FUNCTION_BLOCK "Assembler_devic"   // FB1, GRAPH
{ S7_Optimized_Access := 'FALSE' }
VERSION : 0.1
   VAR_INPUT
      OFF_SQ : Bool := false;   // Turn sequence off
      INIT_SQ : Bool := false;   // Set sequence to initial state
      ACK_EF : Bool := false;   // Acknowledge all errors and faults
      S_PREV : Bool := false;   // Output previous step in parameter S_NO
      S_NEXT : Bool := false;   // Indicate next step in parameter S_NO
      SW_AUTO : Bool := false;   // Automatic mode
      SW_TAP : Bool := false;   // Semiautomatic/switch with transition
      SW_TOP : Bool := false;   // Semiautomatic/ignore transition
      SW_MAN : Bool := false;   // Manual mode
      S_SEL : Int := 0;   // Select step to be output to S_NO
      S_ON : Bool := false;   // Activate step indicated in S_NO
      S_OFF : Bool := false;   // Deactivate step indicated S_NO
      T_PUSH : Bool := false;   // Enable transition to switch in semi automatic mode
   END_VAR
   VAR_OUTPUT
      S_NO : Int := 0;   // Step number
      S_MORE : Bool := false;   // More steps are available and can be shown in S_NO
      S_ACTIVE : Bool := false;   // Step indicated in S_NO is active
      ERR_FLT : Bool := false;   // Interlock or supervision group error
      AUTO_ON : Bool := false;   // Automatic mode is active
      TAP_ON : Bool := false;   // Semiautomatic mode/step with transition enabled
      TOP_ON : Bool := false;   // Semiautomatic mode/ignore transition enabled
      MAN_ON : Bool := false;   // Manual mode is active
   END_VAR
   VAR_IN_OUT
      "assembler x set point" : Real;
      "assembler x set point value" : Real;
      "assembler z set point" : Real;
      "assembler z set point value" : Real;
      "assembler grab" : Bool;
      "assembler grabed" : Bool;
      "lid clamp" : Bool;
      "base clamp" : Bool;
      "lid clamped" : Bool;
      "base clamped" : Bool;
      "base rise" : Bool;
      "base limit" : Bool;
      "line1  ready" : Bool;
      "line2  ready" : Bool;
      "assembler rotate" : Bool;
      "assembler rotating" : Bool;
      "assembler complete" : Bool;
   END_VAR
   VAR
      SWITCH : Array[0..0] of DWord;
      SW_SQTS : Array[0..14] of Byte;
      SW_ADDR : Word := 16#1C;
      G7T_0 : GraphTransition;
      G7S_0 : GraphStep;
      PRE_CRIT : Array[0..0] of DWord;
      POST_CRIT : Array[0..0] of DWord;
      TVX : Array[0..4] of Byte;
      TTX : Array[0..4] of Byte;
      TSX : Array[0..4] of Byte;
      S00X : Array[0..4] of Byte;
      SOFFX : Array[0..4] of Byte;
      SONX : Array[0..4] of Byte;
      SAX : Array[0..4] of Byte;
      SERRX : Array[0..15] of Byte;
      SMX : Array[0..15] of Byte;
      S0X : Array[0..15] of Byte;
      S1X : Array[0..15] of Byte;
      S_DISPLAY : Int;   // Internal display of output parameter S_NO
      S_SEL_OLD : Int;   // Previous value in S_SEL
      S_DISPIDX : Byte;   // Index of the step in S_NO
      T_DISPIDX : Byte;   // Index of the transition displayed in T_NO
      MOPEDGE : Struct
         AUTO : Bool := false;
         MAN : Bool := false;
         TAP : Bool := false;
         TOP : Bool := false;
         ACK_S : Bool := false;
         REG_S : Bool := false;
         T_PREV : Bool := false;
         T_NEXT : Bool := false;
         LOCK : Bool := false;
         SUP : Bool := false;
         ACKREQ : Bool := false;
         SSKIP : Bool := false;
         OFF : Bool := false;
         INIT : Bool := false;
         HALT : Bool := false;
         TMS_HALT : Bool := false;
         OPS_ZERO : Bool := false;
         SACT_DISP : Bool := false;
         SEF_DISP : Bool := false;
         SALL_DISP : Bool := false;
         S_PREV : Bool := false;
         S_NEXT : Bool := false;
         S_SELOK : Bool := false;
         S_ON : Bool := false;
         S_OFF : Bool := false;
         T_PUSH : Bool := false;
         REG : Bool := false;
         ACK : Bool := false;
         IL_PERM : Bool := false;
         T_PERM : Bool := false;
         ILP_MAN : Bool := false;
      END_STRUCT;
      MOP : Struct   // Mode
         AUTO : Bool := true;   // Status: automatic mode
         MAN : Bool := false;   // Status: manual mode
         TAP : Bool := false;   // Status: semi automatic/switch with transition
         TOP : Bool := false;   // Status: semi automatic/ignore transition
         ACK_S : Bool := false;   // Request: acknowledge step at parameter S_NO
         REG_S : Bool := false;   // Request: register step indicated in S_NO
         T_PREV : Bool := false;   // Request: output previous valid transition in T_NO
         T_NEXT : Bool := false;   // Request: output next valid transition in T_NO
         LOCK : Bool := true;   // Status: interlocks activated
         SUP : Bool := true;   // Status: supervisions activated
         ACKREQ : Bool := true;   // Status: acknowledgment required
         SSKIP : Bool := false;   // Status: "Skip steps" enabled
         OFF : Bool := false;   // Request: deactivate all steps
         INIT : Bool := true;   // Request: set sequence to initial state
         HALT : Bool := false;   // Status: sequence halted
         TMS_HALT : Bool := false;   // Status: all internal timers held
         OPS_ZERO : Bool := false;   // Status: set all operands processed with N, L, D instructions to 0
         SACT_DISP : Bool := true;   // Status: display active steps only
         SEF_DISP : Bool := false;   // Status: display only steps with errors and disrupted steps
         SALL_DISP : Bool := false;   // Status: display all steps
         S_PREV : Bool := false;   // Request: output previous step to S_NO
         S_NEXT : Bool := false;   // Request: Output next step at S_NO parameter
         S_SELOK : Bool := false;   // Request: output step number from S_SEL to S_NO
         S_ON : Bool := false;   // Request: activate step indicated in S_NO
         S_OFF : Bool := false;   // Request: deactivate step at parameter S_NO
         T_PUSH : Bool := false;   // Request: transition switching enabled
         REG : Bool := false;   // Request: register all interlock and supervision errors
         ACK : Bool := false;   // Request: acknowledge all interlock and supervision errors
         IL_PERM : Bool := false;   // Status: permanent processing of all interlocks
         T_PERM : Bool := false;   // Status: permanent processing of all transitions
         ILP_MAN : Bool := false;   // Status: permanent processing of all interlocks in manual mode
      END_STRUCT;
      TICKS : Struct   // Clock speeds
         DELTA : Time := T#0ms;   // Time difference between cycles
         OLD : Time := T#0ms;   // 10 ms clock counter value in last cycle
         NEW : Time := T#0ms;   // 10 ms clock counter value in this cycle
      END_STRUCT;
      SQ_FLAGS : Struct   // Sequence bit memory
         ERR_FLT : Bool := false;   // Interlock and supervision group error
         ERROR : Bool := false;   // Interlock group error
         FAULT : Bool := false;   // Supervision group error
         RT_FAIL : Bool := false;   // Runtime error
         NO_SNO : Bool := false;   // Requested step number not found
         NF_OFL : Bool := false;   // Overflow: too many ON or OFF requests
         SA_OFL : Bool := false;   // Overflow: too many steps active
         TV_OFL : Bool := false;   // Overflow: too many valid transitions
         MSG_OFL : Bool := false;   // Overflow: not enough system resources for ALARM_S
         NO_SWI : Bool := false;   // Do not switch in this cycle
         CYC_OP : Bool := false;   // Cyclic execution of the sequence after initialization
         AS_MSG : Bool := true;   // Alarms during runtime enabled or disabled by instruction
         AS_SEND : Bool := false;   // Send alarms from WR_USMSG or only enter in diagnostics buffer
         SQ_BUSY : Bool := false;   // Internal edge bit memory for sequence processing
         SA_BUSY : Bool := false;   // Internal edge bit memory for sequence processing
         AS_SIG : Bool := false;   // Edge bit memory for alarms from Alarm_S and Alarm_SQ
      END_STRUCT;
      S_PTR : DWord := 16#890;
      S_PTR2 : DWord := 16#0;
      S_PTR3 : DWord := 16#1AA0;
      S_PTR4 : DWord := 16#1A20;
      T_PTR : DWord := 16#19A0;
      C_AR2 : DWord := 16#0;
      M_FBDB : DWord := 16#10000;
      M_SNO : Word := 16#0;
      M_EVID : Word := 16#0;
      M_EVIL : C_Alarm_s;
      M_EVSV : C_Alarm_s;
      M_EV : DWord := 16#1890;
      CRIT : Array[0..31] of Bool;
      S_START : Byte := 16#0;
      S_IDX : Byte := 16#0;
      S_INT : Int := 72;
      S_TMP : Byte := 16#0;
      T_START : Byte := 16#0;
      T_IDX : Byte := 16#0;
      T_TMP : Byte := 16#0;
      T_TMP2 : Byte := 16#00;
      TV_POT : Byte := 16#06;
      RETURN1 : Byte := 16#0;
      RETURN2 : Byte := 16#0;
      SINI : Array[0..4] of Byte;
      LSTT : Array[0..13] of Byte;
      ATAJ : Array[0..13] of Byte;
      ATAB : Array[0..13] of Byte;
      PSTT : Array[0..13] of Byte;
      NSTT : Array[0..13] of Byte;
      ASSJ : Array[0..14] of Byte;
      ASSB : Array[0..14] of Byte;
      PTTS : Array[0..14] of Byte;
      NTTS : Array[0..14] of Byte;
      PRE_CNT : Word := 16#1;
      POST_CNT : Word := 16#1;
      ADR_COND : Word := 16#0;
      MAX_TVAL : Byte := 16#3;
      MAX_SACT : Byte := 16#3;
      MAX_CRIT : Byte := 16#4;
      T_CNT : Byte := 16#D;
      SUP_CNT : Byte := 16#0;
      LOCK_CNT : Byte;
      S_CNT : Byte := 16#E;
      SQ_CNT : Byte := 16#1;
      PRS_INPAR : DWord := 16#E000FEC8;
      PRS_OUTPAR : DWord := 16#E000800F;
      GC_FLAGS : Struct
         T_MACH : Byte := 16#EB;
         COND_ED : Byte := 16#E3;
         W_LEVEL : Byte := 16#D5;
         FB_IF : Byte := 16#FA;
         AS_MSG : Word := 16#404;
         SSB : Word := 16#108;
         DILG : Word := 16#470;
         ADDR_T0 : Word := 16#32;
         CRIT_AVAIL : Bool := false;
         SSKIP_AVAIL : Bool := true;
         SSKIP_ON : Bool := false;
         ACK_REQ : Bool := true;
         SYNC_AVAIL : Bool := true;
         ILP_MAN : Bool := false;
         SWM_LOCKED : Bool := false;
         SAVE_SW : Bool := true;
      END_STRUCT;
      G7_FBMARK : Byte := 16#3C;
      G7_RELEASE : Byte := 16#3C;
      G7_ID2 : Byte := 16#37;
      G7_ID1 : Byte := 16#47;
   END_VAR
   // SW_SQTS[0] := 16#4;
   // SWITCH[0] := 16#40020000;
   // SW_SQTS[2] := 16#1;
   // SW_SQTS[3] := 16#1;
   // SW_SQTS[4] := 16#2;
   // SW_SQTS[5] := 16#2;
   // SW_SQTS[6] := 16#2;
   // SW_SQTS[7] := 16#3;
   // TVX[0] := 16#1;
   // TTX[0] := 16#1;
   // TSX[0] := 16#1;
   // S00X[0] := 16#1;
   // SOFFX[0] := 16#1;
   // SONX[0] := 16#1;
   // SAX[0] := 16#1;
   // SERRX[0] := 16#1;
   // SMX[0] := 16#1;
   // S0X[0] := 16#1;
   // S1X[0] := 16#1;
   // SINI[0] := 16#2;
   // SINI[1] := 16#1;
   // SINI[2] := 0;
   // SINI[3] := 0;
   // SINI[4] := 0;
   // LSTT[0] := 0;
   // LSTT[1] := 0;
   // LSTT[2] := 0;
   // LSTT[3] := 0;
   // LSTT[4] := 0;
   // LSTT[5] := 0;
   // LSTT[6] := 0;
   // LSTT[7] := 0;
   // ATAJ[0] := 0;
   // ATAJ[1] := 16#1;
   // ATAJ[2] := 16#2;
   // ATAJ[3] := 16#3;
   // ATAJ[4] := 16#4;
   // ATAJ[5] := 16#5;
   // ATAJ[6] := 16#6;
   // ATAJ[7] := 16#7;
   // ATAB[0] := 0;
   // ATAB[1] := 16#1;
   // ATAB[2] := 16#2;
   // ATAB[3] := 16#3;
   // ATAB[4] := 16#4;
   // ATAB[5] := 16#5;
   // ATAB[6] := 16#6;
   // ATAB[7] := 16#7;
   // PSTT[0] := 0;
   // PSTT[1] := 16#1;
   // PSTT[2] := 16#2;
   // PSTT[3] := 16#3;
   // PSTT[4] := 16#4;
   // PSTT[5] := 16#5;
   // PSTT[6] := 16#8;
   // PSTT[7] := 16#9;
   // NSTT[0] := 16#1;
   // NSTT[1] := 16#2;
   // NSTT[2] := 16#3;
   // NSTT[3] := 16#8;
   // NSTT[5] := 16#6;
   // NSTT[6] := 16#9;
   // NSTT[7] := 16#A;
   // ASSJ[0] := 0;
   // ASSJ[1] := 16#1;
   // ASSJ[2] := 16#2;
   // ASSJ[3] := 16#6;
   // ASSJ[4] := 16#4;
   // ASSJ[5] := 16#5;
   // ASSJ[6] := 16#3;
   // ASSJ[7] := 16#7;
   // ASSB[0] := 0;
   // ASSB[1] := 16#1;
   // ASSB[2] := 16#4;
   // ASSB[3] := 16#3;
   // ASSB[4] := 16#2;
   // ASSB[5] := 16#5;
   // ASSB[6] := 16#6;
   // ASSB[7] := 16#7;
   // PTTS[0] := 0;
   // PTTS[2] := 16#1;
   // PTTS[3] := 16#2;
   // PTTS[4] := 16#1;
   // PTTS[5] := 16#4;
   // PTTS[6] := 16#5;
   // PTTS[7] := 16#8;
   // NTTS[0] := 0;
   // NTTS[1] := 16#1;
   // NTTS[2] := 16#2;
   // NTTS[3] := 16#3;
   // NTTS[4] := 16#4;
   // NTTS[5] := 16#5;
   // NTTS[6] := 16#3;
   // NTTS[7] := 16#9;
   // SW_SQTS[8] := 16#3;
   // NTTS[14] := 16#D;
   // PTTS[14] := 16#C;
   // PTTS[13] := 16#B;
   // ASSB[14] := 16#E;
   // ASSB[13] := 16#D;
   // ASSJ[14] := 16#E;
   // ASSJ[13] := 16#D;
   // NSTT[13] := 16#1;
   // NSTT[12] := 16#E;
   // PSTT[13] := 16#E;
   // ATAB[13] := 16#D;
   // ATAB[12] := 16#C;
   // ATAJ[13] := 16#D;
   // ATAJ[12] := 16#C;
   // LSTT[13] := 16#1;
   // LSTT[12] := 0;
   // SW_SQTS[14] := 16#3;
   // SW_SQTS[13] := 16#3;
   // NSTT[4] := 16#5;
   // NTTS[12] := 16#B;
   // NTTS[11] := 16#A;
   // NTTS[10] := 16#8;
   // NTTS[9] := 16#7;
   // PTTS[12] := 16#A;
   // PTTS[11] := 16#9;
   // PTTS[10] := 16#7;
   // ASSJ[8] := 16#8;
   // ASSB[12] := 16#C;
   // ASSB[11] := 16#B;
   // ASSB[10] := 16#A;
   // ASSB[9] := 16#9;
   // ASSJ[12] := 16#C;
   // ASSJ[11] := 16#B;
   // ASSJ[10] := 16#A;
   // ASSJ[9] := 16#9;
   // NSTT[11] := 16#D;
   // ASSB[8] := 16#8;
   // NSTT[9] := 16#B;
   // NSTT[8] := 16#7;
   // PSTT[11] := 16#C;
   // PSTT[10] := 16#B;
   // PSTT[9] := 16#7;
   // PSTT[8] := 16#A;
   // ATAB[11] := 16#B;
   // ATAB[10] := 16#A;
   // ATAB[9] := 16#9;
   // PTTS[8] := 16#3;
   // ATAJ[11] := 16#B;
   // ATAJ[10] := 16#A;
   // ATAJ[9] := 16#9;
   // ATAJ[8] := 16#8;
   // LSTT[11] := 0;
   // LSTT[10] := 0;
   // LSTT[9] := 0;
   // LSTT[8] := 0;
   // SW_SQTS[12] := 16#3;
   // NTTS[8] := 16#6;
   // SW_SQTS[10] := 16#3;
   // SW_SQTS[9] := 16#3;
   // ATAB[8] := 16#8;
   // NSTT[10] := 16#C;
   // PTTS[9] := 16#6;
   // PSTT[12] := 16#D;
   // NTTS[13] := 16#C;
   // SW_SQTS[11] := 16#3;
BEGIN
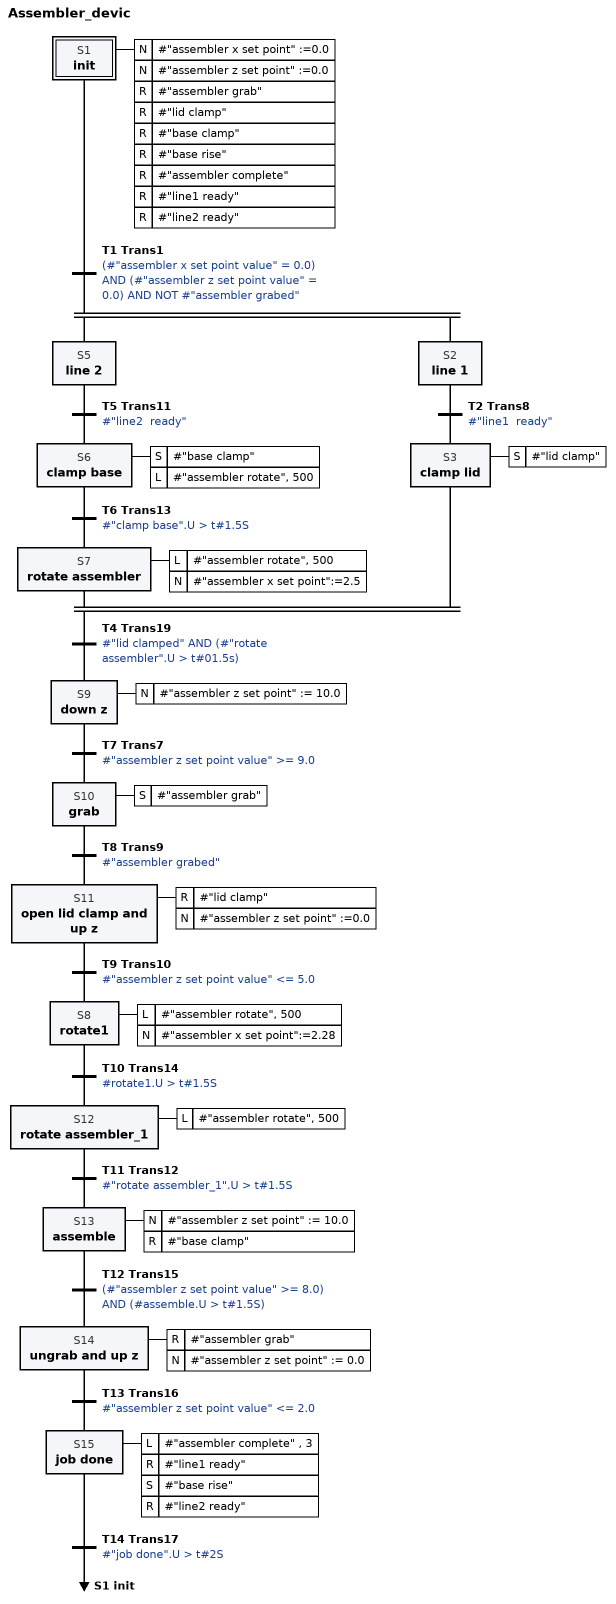
   // sequencer 1
   INITIAL_STEP init:   // S1
              N    #"assembler x set point" :=0.0
              N    #"assembler z set point" :=0.0
              R    #"assembler grab"
              R    #"lid clamp"
              R    #"base clamp"
              R    #"base rise"
              R    #"assembler complete"
              R    #"line1  ready"
              R    #"line2  ready"
   END_STEP
   TRANSITION Trans1 FROM init TO ("line 2", "line 1")   // T1
      := (#"assembler x set point value" = 0.0) AND (#"assembler z set point value" = 0.0) AND NOT #"assembler grabed";
   END_TRANSITION
   STEP "clamp lid":   // S3
              S    #"lid clamp"
   END_STEP
   STEP "line 2":   // S5
   END_STEP
   TRANSITION Trans11 FROM "line 2" TO "clamp base"   // T5
      := #"line2  ready";
   END_TRANSITION
   STEP "line 1":   // S2
   END_STEP
   TRANSITION Trans8 FROM "line 1" TO "clamp lid"   // T2
      := #"line1  ready";
   END_TRANSITION
   STEP grab:   // S10
              S    #"assembler grab"
   END_STEP
   TRANSITION Trans9 FROM grab TO "open lid clamp and up z"   // T8
      := #"assembler grabed";
   END_TRANSITION
   STEP "clamp base":   // S6
              S    #"base clamp"
              L    #"assembler rotate", 500
   END_STEP
   TRANSITION Trans13 FROM "clamp base" TO "rotate assembler"   // T6
      := #"clamp base".U > t#1.5S;
   END_TRANSITION
   STEP "rotate assembler":   // S7
              L    #"assembler rotate", 500
              N    #"assembler x set point":=2.5
   END_STEP
   TRANSITION Trans19 FROM ("clamp lid", "rotate assembler") TO "down z"   // T4
      := #"lid clamped" AND (#"rotate assembler".U > t#01.5s);
   END_TRANSITION
   STEP "down z":   // S9
              N    #"assembler z set point" := 10.0
   END_STEP
   TRANSITION Trans7 FROM "down z" TO grab   // T7
      := #"assembler z set point value" >= 9.0;
   END_TRANSITION
   STEP "open lid clamp and up z":   // S11
              R    #"lid clamp"
              N    #"assembler z set point" :=0.0
   END_STEP
   TRANSITION Trans10 FROM "open lid clamp and up z" TO rotate1   // T9
      := #"assembler z set point value" <= 5.0;
   END_TRANSITION
   STEP rotate1:   // S8
              L    #"assembler rotate", 500
              N    #"assembler x set point":=2.28
   END_STEP
   TRANSITION Trans14 FROM rotate1 TO "rotate assembler_1"   // T10
      := #rotate1.U > t#1.5S;
   END_TRANSITION
   STEP "rotate assembler_1":   // S12
              L    #"assembler rotate", 500
   END_STEP
   TRANSITION Trans12 FROM "rotate assembler_1" TO assemble   // T11
      := #"rotate assembler_1".U > t#1.5S;
   END_TRANSITION
   STEP assemble:   // S13
              N    #"assembler z set point" := 10.0
              R    #"base clamp"
   END_STEP
   TRANSITION Trans15 FROM assemble TO "ungrab and up z"   // T12
      := (#"assembler z set point value" >= 8.0) AND (#assemble.U > t#1.5S);
   END_TRANSITION
   STEP "ungrab and up z":   // S14
              R    #"assembler grab"
              N    #"assembler z set point" := 0.0
   END_STEP
   TRANSITION Trans16 FROM "ungrab and up z" TO "job done"   // T13
      := #"assembler z set point value" <= 2.0;
   END_TRANSITION
   STEP "job done":   // S15
              L    #"assembler complete" , 3
              R    #"line1  ready"
              S    #"base rise"
              R    #"line2  ready"
   END_STEP
   TRANSITION Trans17 FROM "job done" TO init   // T14, jump
      := #"job done".U > t#2S;
   END_TRANSITION
END_FUNCTION_BLOCK

FUNCTION "Assembler" : Void   // FC4, LAD
{ S7_Optimized_Access := 'FALSE' }
VERSION : 0.1
BEGIN

REGION Network 1: Control Convoyers
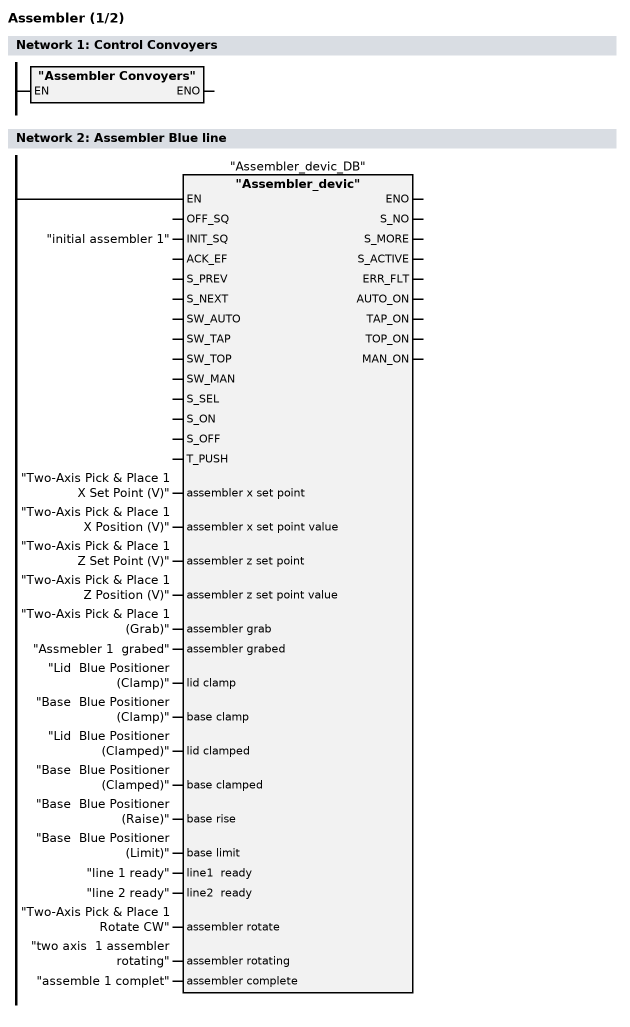
   RUNG wire#powerrail
      "Assembler Convoyers"()
   END_RUNG
   // the same network as SCL:
   "Assembler Convoyers"();
END_REGION

REGION Network 2: Assembler Blue line
   RUNG wire#powerrail
      "Assembler_devic_DB"(OFF_SQ :=, INIT_SQ := "initial assembler 1", ACK_EF :=, S_PREV :=, S_NEXT :=, SW_AUTO :=, SW_TAP :=, SW_TOP :=, SW_MAN :=, S_SEL :=, S_ON :=, S_OFF :=, T_PUSH :=, "assembler x set point" := "Two-Axis Pick & Place 1 X Set Point (V)", "assembler x set point value" := "Two-Axis Pick & Place 1 X Position (V)", "assembler z set point" := "Two-Axis Pick & Place 1 Z Set Point (V)", "assembler z set point value" := "Two-Axis Pick & Place 1 Z Position (V)", "assembler grab" := "Two-Axis Pick & Place 1 (Grab)", "assembler grabed" := "Assmebler 1  grabed", "lid clamp" := "Lid  Blue Positioner (Clamp)", "base clamp" := "Base  Blue Positioner (Clamp)", "lid clamped" := "Lid  Blue Positioner (Clamped)", "base clamped" := "Base  Blue Positioner (Clamped)", "base rise" := "Base  Blue Positioner  (Raise)", "base limit" := "Base  Blue Positioner (Limit)", "line1  ready" := "line 1 ready", "line2  ready" := "line 2 ready", "assembler rotate" := "Two-Axis Pick & Place 1 Rotate CW", "assembler rotating" := "two axis  1 assembler rotating", "assembler complete" := "assemble 1 complet", S_NO =>, S_MORE =>, S_ACTIVE =>, ERR_FLT =>, AUTO_ON =>, TAP_ON =>, TOP_ON =>, MAN_ON =>)
   END_RUNG
   // the same network as SCL:
   "Assembler_devic_DB"(INIT_SQ := "initial assembler 1",   // "Assembler_devic"
                        "assembler x set point" := "Two-Axis Pick & Place 1 X Set Point (V)",
                        "assembler x set point value" := "Two-Axis Pick & Place 1 X Position (V)",
                        "assembler z set point" := "Two-Axis Pick & Place 1 Z Set Point (V)",
                        "assembler z set point value" := "Two-Axis Pick & Place 1 Z Position (V)",
                        "assembler grab" := "Two-Axis Pick & Place 1 (Grab)",
                        "assembler grabed" := "Assmebler 1  grabed",
                        "lid clamp" := "Lid  Blue Positioner (Clamp)",
                        "base clamp" := "Base  Blue Positioner (Clamp)",
                        "lid clamped" := "Lid  Blue Positioner (Clamped)",
                        "base clamped" := "Base  Blue Positioner (Clamped)",
                        "base rise" := "Base  Blue Positioner  (Raise)",
                        "base limit" := "Base  Blue Positioner (Limit)",
                        "line1  ready" := "line 1 ready",
                        "line2  ready" := "line 2 ready",
                        "assembler rotate" := "Two-Axis Pick & Place 1 Rotate CW",
                        "assembler rotating" := "two axis  1 assembler rotating",
                        "assembler complete" := "assemble 1 complet");
END_REGION

REGION Network 3: Assembler green line
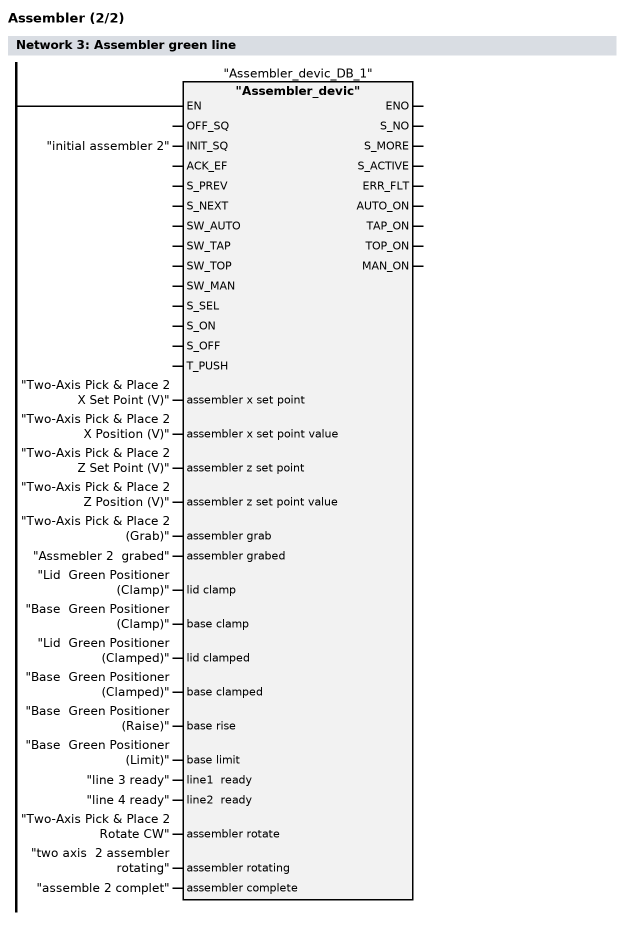
   RUNG wire#powerrail
      "Assembler_devic_DB_1"(OFF_SQ :=, INIT_SQ := "initial assembler 2", ACK_EF :=, S_PREV :=, S_NEXT :=, SW_AUTO :=, SW_TAP :=, SW_TOP :=, SW_MAN :=, S_SEL :=, S_ON :=, S_OFF :=, T_PUSH :=, "assembler x set point" := "Two-Axis Pick & Place 2 X Set Point (V)", "assembler x set point value" := "Two-Axis Pick & Place 2 X Position (V)", "assembler z set point" := "Two-Axis Pick & Place 2 Z Set Point (V)", "assembler z set point value" := "Two-Axis Pick & Place 2 Z Position (V)", "assembler grab" := "Two-Axis Pick & Place 2 (Grab)", "assembler grabed" := "Assmebler 2  grabed", "lid clamp" := "Lid  Green Positioner (Clamp)", "base clamp" := "Base  Green Positioner (Clamp)", "lid clamped" := "Lid  Green Positioner (Clamped)", "base clamped" := "Base  Green Positioner (Clamped)", "base rise" := "Base  Green Positioner (Raise)", "base limit" := "Base  Green Positioner (Limit)", "line1  ready" := "line 3 ready", "line2  ready" := "line 4 ready", "assembler rotate" := "Two-Axis Pick & Place 2 Rotate CW", "assembler rotating" := "two axis  2 assembler rotating", "assembler complete" := "assemble 2 complet", S_NO =>, S_MORE =>, S_ACTIVE =>, ERR_FLT =>, AUTO_ON =>, TAP_ON =>, TOP_ON =>, MAN_ON =>)
   END_RUNG
   // the same network as SCL:
   "Assembler_devic_DB_1"(INIT_SQ := "initial assembler 2",   // "Assembler_devic"
                          "assembler x set point" := "Two-Axis Pick & Place 2 X Set Point (V)",
                          "assembler x set point value" := "Two-Axis Pick & Place 2 X Position (V)",
                          "assembler z set point" := "Two-Axis Pick & Place 2 Z Set Point (V)",
                          "assembler z set point value" := "Two-Axis Pick & Place 2 Z Position (V)",
                          "assembler grab" := "Two-Axis Pick & Place 2 (Grab)",
                          "assembler grabed" := "Assmebler 2  grabed",
                          "lid clamp" := "Lid  Green Positioner (Clamp)",
                          "base clamp" := "Base  Green Positioner (Clamp)",
                          "lid clamped" := "Lid  Green Positioner (Clamped)",
                          "base clamped" := "Base  Green Positioner (Clamped)",
                          "base rise" := "Base  Green Positioner (Raise)",
                          "base limit" := "Base  Green Positioner (Limit)",
                          "line1  ready" := "line 3 ready",
                          "line2  ready" := "line 4 ready",
                          "assembler rotate" := "Two-Axis Pick & Place 2 Rotate CW",
                          "assembler rotating" := "two axis  2 assembler rotating",
                          "assembler complete" := "assemble 2 complet");
END_REGION
END_FUNCTION

FUNCTION "Sort" : Void   // FC5, LAD
{ S7_Optimized_Access := 'FALSE' }
VERSION : 0.1
BEGIN

REGION Network 1: Blue Lid
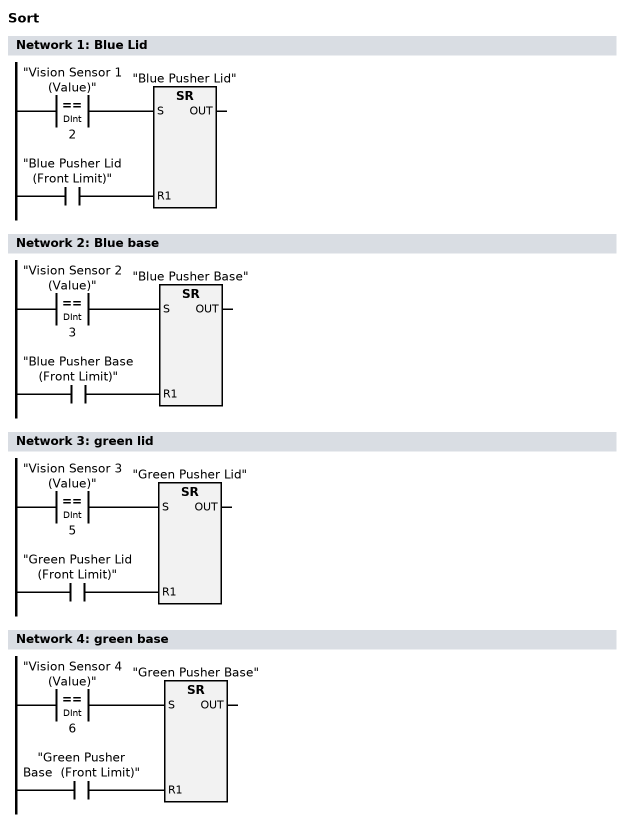
   RUNG wire#powerrail
      { S7_Templates := "SrcType := DInt" } EQ_Contact(in1 := "Vision Sensor 1 (Value)", in2 := 2)
      S_SR(operand := "Blue Pusher Lid", r1 := wire#w1)
   END_RUNG
   RUNG wire#powerrail
      Contact( "Blue Pusher Lid (Front Limit)" )
   END_RUNG wire#w1
   // the same network as SCL:
   IF "Vision Sensor 1 (Value)" = 2 THEN
       "Blue Pusher Lid" := TRUE;   // SR flip-flop
   END_IF;
   IF "Blue Pusher Lid (Front Limit)" THEN "Blue Pusher Lid" := FALSE; END_IF;
END_REGION

REGION Network 2: Blue base
   RUNG wire#powerrail
      { S7_Templates := "SrcType := DInt" } EQ_Contact(in1 := "Vision Sensor 2 (Value)", in2 := 3)
      S_SR(operand := "Blue Pusher Base", r1 := wire#w1)
   END_RUNG
   RUNG wire#powerrail
      Contact( "Blue Pusher Base  (Front Limit)" )
   END_RUNG wire#w1
   // the same network as SCL:
   IF "Vision Sensor 2 (Value)" = 3 THEN
       "Blue Pusher Base" := TRUE;   // SR flip-flop
   END_IF;
   IF "Blue Pusher Base  (Front Limit)" THEN "Blue Pusher Base" := FALSE; END_IF;
END_REGION

REGION Network 3: green lid
   RUNG wire#powerrail
      { S7_Templates := "SrcType := DInt" } EQ_Contact(in1 := "Vision Sensor 3 (Value)", in2 := 5)
      S_SR(operand := "Green Pusher Lid", r1 := wire#w1)
   END_RUNG
   RUNG wire#powerrail
      Contact( "Green Pusher Lid (Front Limit)" )
   END_RUNG wire#w1
   // the same network as SCL:
   IF "Vision Sensor 3 (Value)" = 5 THEN
       "Green Pusher Lid" := TRUE;   // SR flip-flop
   END_IF;
   IF "Green Pusher Lid (Front Limit)" THEN "Green Pusher Lid" := FALSE; END_IF;
END_REGION

REGION Network 4: green base
   RUNG wire#powerrail
      { S7_Templates := "SrcType := DInt" } EQ_Contact(in1 := "Vision Sensor 4 (Value)", in2 := 6)
      S_SR(operand := "Green Pusher Base", r1 := wire#w1)
   END_RUNG
   RUNG wire#powerrail
      Contact( "Green Pusher Base  (Front Limit)" )
   END_RUNG wire#w1
   // the same network as SCL:
   IF "Vision Sensor 4 (Value)" = 6 THEN
       "Green Pusher Base" := TRUE;   // SR flip-flop
   END_IF;
   IF "Green Pusher Base  (Front Limit)" THEN "Green Pusher Base" := FALSE; END_IF;
END_REGION
END_FUNCTION

FUNCTION "Assembler Convoyers" : Void   // FC6, LAD
{ S7_Optimized_Access := 'FALSE' }
VERSION : 0.1
   VAR_TEMP   // added for the SCL form of the ladder/FBD networks
      _w1 : Bool;
      _w2 : Bool;
      _w3 : Bool;
   END_VAR
BEGIN

REGION Network 1: Blue lid Convoyer *
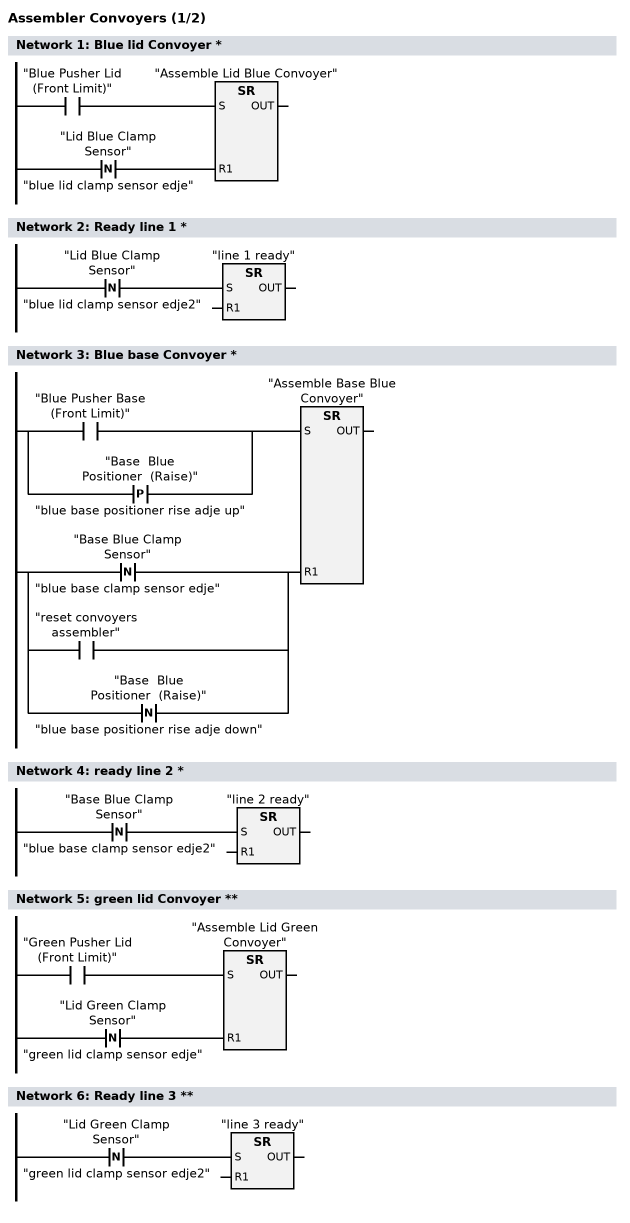
   RUNG wire#powerrail
      Contact( "Blue Pusher Lid (Front Limit)" )
      S_SR(operand := "Assemble Lid Blue Convoyer", r1 := wire#w1)
   END_RUNG
   RUNG wire#powerrail
      N_Contact(operand := "Lid Blue Clamp Sensor", bit := "blue lid clamp sensor edje")
   END_RUNG wire#w1
   // the same network as SCL:
   #_w1 := NOT "Lid Blue Clamp Sensor" AND "blue lid clamp sensor edje";   // falling edge of "Lid Blue Clamp Sensor"
   "blue lid clamp sensor edje" := "Lid Blue Clamp Sensor";
   IF "Blue Pusher Lid (Front Limit)" THEN
       "Assemble Lid Blue Convoyer" := TRUE;   // SR flip-flop
   END_IF;
   IF #_w1 THEN "Assemble Lid Blue Convoyer" := FALSE; END_IF;
END_REGION

REGION Network 2: Ready line 1 *
   RUNG wire#powerrail
      N_Contact(operand := "Lid Blue Clamp Sensor", bit := "blue lid clamp sensor edje2")
      S_SR(operand := "line 1 ready", r1 :=)
   END_RUNG
   // the same network as SCL:
   #_w1 := NOT "Lid Blue Clamp Sensor" AND "blue lid clamp sensor edje2";   // falling edge of "Lid Blue Clamp Sensor"
   "blue lid clamp sensor edje2" := "Lid Blue Clamp Sensor";
   IF #_w1 THEN
       "line 1 ready" := TRUE;   // SR flip-flop
   END_IF;
END_REGION

REGION Network 3: Blue base Convoyer *
   RUNG wire#powerrail
      Contact( "Blue Pusher Base  (Front Limit)" )
      wire#w1
      S_SR(operand := "Assemble Base Blue Convoyer", r1 := wire#w2)
   END_RUNG
   RUNG wire#powerrail
      P_Contact(operand := "Base  Blue Positioner  (Raise)", bit := "blue base positioner rise adje up")
   END_RUNG wire#w1
   RUNG wire#powerrail
      N_Contact(operand := "Base Blue Clamp Sensor", bit := "blue base clamp sensor edje")
   END_RUNG wire#w2
   RUNG wire#powerrail
      Contact( "reset convoyers assembler" )
   END_RUNG wire#w2
   RUNG wire#powerrail
      N_Contact(operand := "Base  Blue Positioner  (Raise)", bit := "blue base positioner rise adje down")
   END_RUNG wire#w2
   // the same network as SCL:
   #_w1 := "Base  Blue Positioner  (Raise)" AND NOT "blue base positioner rise adje up";   // rising edge of "Base  Blue Positioner  (Raise)"
   "blue base positioner rise adje up" := "Base  Blue Positioner  (Raise)";
   #_w2 := NOT "Base Blue Clamp Sensor" AND "blue base clamp sensor edje";   // falling edge of "Base Blue Clamp Sensor"
   "blue base clamp sensor edje" := "Base Blue Clamp Sensor";
   #_w3 := NOT "Base  Blue Positioner  (Raise)" AND "blue base positioner rise adje down";   // falling edge of "Base  Blue Positioner  (Raise)"
   "blue base positioner rise adje down" := "Base  Blue Positioner  (Raise)";
   IF "Blue Pusher Base  (Front Limit)" OR #_w1 THEN
       "Assemble Base Blue Convoyer" := TRUE;   // SR flip-flop
   END_IF;
   IF #_w2 OR "reset convoyers assembler" OR #_w3 THEN "Assemble Base Blue Convoyer" := FALSE; END_IF;
END_REGION

REGION Network 4: ready line 2 *
   RUNG wire#powerrail
      N_Contact(operand := "Base Blue Clamp Sensor", bit := "blue base clamp sensor edje2")
      S_SR(operand := "line 2 ready", r1 :=)
   END_RUNG
   // the same network as SCL:
   #_w1 := NOT "Base Blue Clamp Sensor" AND "blue base clamp sensor edje2";   // falling edge of "Base Blue Clamp Sensor"
   "blue base clamp sensor edje2" := "Base Blue Clamp Sensor";
   IF #_w1 THEN
       "line 2 ready" := TRUE;   // SR flip-flop
   END_IF;
END_REGION

REGION Network 5: green lid Convoyer **
   RUNG wire#powerrail
      Contact( "Green Pusher Lid (Front Limit)" )
      S_SR(operand := "Assemble Lid Green Convoyer", r1 := wire#w1)
   END_RUNG
   RUNG wire#powerrail
      N_Contact(operand := "Lid Green Clamp Sensor", bit := "green lid clamp sensor edje")
   END_RUNG wire#w1
   // the same network as SCL:
   #_w1 := NOT "Lid Green Clamp Sensor" AND "green lid clamp sensor edje";   // falling edge of "Lid Green Clamp Sensor"
   "green lid clamp sensor edje" := "Lid Green Clamp Sensor";
   IF "Green Pusher Lid (Front Limit)" THEN
       "Assemble Lid Green Convoyer" := TRUE;   // SR flip-flop
   END_IF;
   IF #_w1 THEN "Assemble Lid Green Convoyer" := FALSE; END_IF;
END_REGION

REGION Network 6: Ready line 3 **
   RUNG wire#powerrail
      N_Contact(operand := "Lid Green Clamp Sensor", bit := "green lid clamp sensor edje2")
      S_SR(operand := "line 3 ready", r1 :=)
   END_RUNG
   // the same network as SCL:
   #_w1 := NOT "Lid Green Clamp Sensor" AND "green lid clamp sensor edje2";   // falling edge of "Lid Green Clamp Sensor"
   "green lid clamp sensor edje2" := "Lid Green Clamp Sensor";
   IF #_w1 THEN
       "line 3 ready" := TRUE;   // SR flip-flop
   END_IF;
END_REGION

REGION Network 7: green base Convoyer **
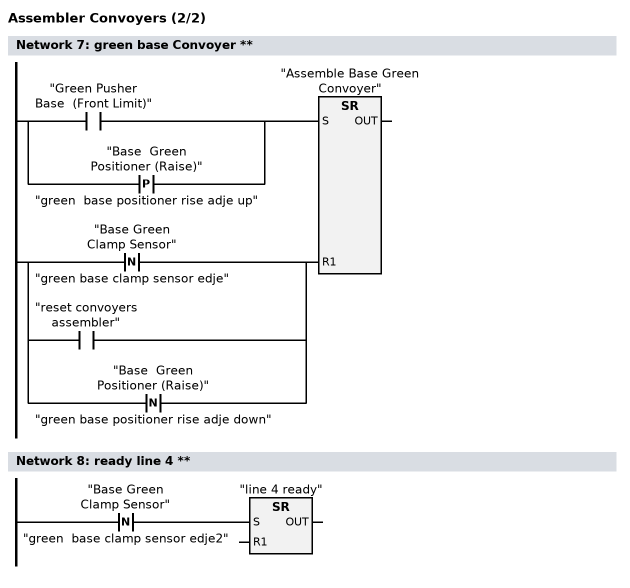
   RUNG wire#powerrail
      Contact( "Green Pusher Base  (Front Limit)" )
      wire#w1
      S_SR(operand := "Assemble Base Green Convoyer", r1 := wire#w2)
   END_RUNG
   RUNG wire#powerrail
      P_Contact(operand := "Base  Green Positioner (Raise)", bit := "green  base positioner rise adje up")
   END_RUNG wire#w1
   RUNG wire#powerrail
      N_Contact(operand := "Base Green Clamp Sensor", bit := "green base clamp sensor edje")
   END_RUNG wire#w2
   RUNG wire#powerrail
      Contact( "reset convoyers assembler" )
   END_RUNG wire#w2
   RUNG wire#powerrail
      N_Contact(operand := "Base  Green Positioner (Raise)", bit := "green base positioner rise adje down")
   END_RUNG wire#w2
   // the same network as SCL:
   #_w1 := "Base  Green Positioner (Raise)" AND NOT "green  base positioner rise adje up";   // rising edge of "Base  Green Positioner (Raise)"
   "green  base positioner rise adje up" := "Base  Green Positioner (Raise)";
   #_w2 := NOT "Base Green Clamp Sensor" AND "green base clamp sensor edje";   // falling edge of "Base Green Clamp Sensor"
   "green base clamp sensor edje" := "Base Green Clamp Sensor";
   #_w3 := NOT "Base  Green Positioner (Raise)" AND "green base positioner rise adje down";   // falling edge of "Base  Green Positioner (Raise)"
   "green base positioner rise adje down" := "Base  Green Positioner (Raise)";
   IF "Green Pusher Base  (Front Limit)" OR #_w1 THEN
       "Assemble Base Green Convoyer" := TRUE;   // SR flip-flop
   END_IF;
   IF #_w2 OR "reset convoyers assembler" OR #_w3 THEN "Assemble Base Green Convoyer" := FALSE; END_IF;
END_REGION

REGION Network 8: ready line 4 **
   RUNG wire#powerrail
      N_Contact(operand := "Base Green Clamp Sensor", bit := "green  base clamp sensor edje2")
      S_SR(operand := "line 4 ready", r1 :=)
   END_RUNG
   // the same network as SCL:
   #_w1 := NOT "Base Green Clamp Sensor" AND "green  base clamp sensor edje2";   // falling edge of "Base Green Clamp Sensor"
   "green  base clamp sensor edje2" := "Base Green Clamp Sensor";
   IF #_w1 THEN
       "line 4 ready" := TRUE;   // SR flip-flop
   END_IF;
END_REGION
END_FUNCTION

// folder: Storage System

FUNCTION_BLOCK "Turntable"   // FB4, GRAPH
{ S7_Optimized_Access := 'FALSE' }
VERSION : 0.1
   VAR_INPUT
      OFF_SQ : Bool := false;   // Turn sequence off
      INIT_SQ : Bool := false;   // Set sequence to initial state
      ACK_EF : Bool := false;   // Acknowledge all errors and faults
      S_PREV : Bool := false;   // Output previous step in parameter S_NO
      S_NEXT : Bool := false;   // Indicate next step in parameter S_NO
      SW_AUTO : Bool := false;   // Automatic mode
      SW_TAP : Bool := false;   // Semiautomatic/switch with transition
      SW_TOP : Bool := false;   // Semiautomatic/ignore transition
      SW_MAN : Bool := false;   // Manual mode
      S_SEL : Int := 0;   // Select step to be output to S_NO
      S_ON : Bool := false;   // Activate step indicated in S_NO
      S_OFF : Bool := false;   // Deactivate step indicated S_NO
      T_PUSH : Bool := false;   // Enable transition to switch in semi automatic mode
   END_VAR
   VAR_OUTPUT
      S_NO : Int := 0;   // Step number
      S_MORE : Bool := false;   // More steps are available and can be shown in S_NO
      S_ACTIVE : Bool := false;   // Step indicated in S_NO is active
      ERR_FLT : Bool := false;   // Interlock or supervision group error
      AUTO_ON : Bool := false;   // Automatic mode is active
      TAP_ON : Bool := false;   // Semiautomatic mode/step with transition enabled
      TOP_ON : Bool := false;   // Semiautomatic mode/ignore transition enabled
      MAN_ON : Bool := false;   // Manual mode is active
   END_VAR
   VAR
      SWITCH : Array[0..1] of DWord;
      SW_SQTS : Array[0..15] of Byte;
      SW_ADDR : Word := 16#A;
      G7T_0 : GraphTransition;
      G7S_0 : GraphStep;
      PRE_CRIT : Array[0..0] of DWord;
      POST_CRIT : Array[0..0] of DWord;
      TVX : Array[0..7] of Byte;
      TTX : Array[0..7] of Byte;
      TSX : Array[0..2] of Byte;
      S00X : Array[0..2] of Byte;
      SOFFX : Array[0..2] of Byte;
      SONX : Array[0..2] of Byte;
      SAX : Array[0..2] of Byte;
      SERRX : Array[0..16] of Byte;
      SMX : Array[0..16] of Byte;
      S0X : Array[0..16] of Byte;
      S1X : Array[0..16] of Byte;
      S_DISPLAY : Int;   // Internal display of output parameter S_NO
      S_SEL_OLD : Int;   // Previous value in S_SEL
      S_DISPIDX : Byte;   // Index of the step in S_NO
      T_DISPIDX : Byte;   // Index of the transition displayed in T_NO
      MOPEDGE : Struct
         AUTO : Bool := false;
         MAN : Bool := false;
         TAP : Bool := false;
         TOP : Bool := false;
         ACK_S : Bool := false;
         REG_S : Bool := false;
         T_PREV : Bool := false;
         T_NEXT : Bool := false;
         LOCK : Bool := false;
         SUP : Bool := false;
         ACKREQ : Bool := false;
         SSKIP : Bool := false;
         OFF : Bool := false;
         INIT : Bool := false;
         HALT : Bool := false;
         TMS_HALT : Bool := false;
         OPS_ZERO : Bool := false;
         SACT_DISP : Bool := false;
         SEF_DISP : Bool := false;
         SALL_DISP : Bool := false;
         S_PREV : Bool := false;
         S_NEXT : Bool := false;
         S_SELOK : Bool := false;
         S_ON : Bool := false;
         S_OFF : Bool := false;
         T_PUSH : Bool := false;
         REG : Bool := false;
         ACK : Bool := false;
         IL_PERM : Bool := false;
         T_PERM : Bool := false;
         ILP_MAN : Bool := false;
      END_STRUCT;
      MOP : Struct   // Mode
         AUTO : Bool := true;   // Status: automatic mode
         MAN : Bool := false;   // Status: manual mode
         TAP : Bool := false;   // Status: semi automatic/switch with transition
         TOP : Bool := false;   // Status: semi automatic/ignore transition
         ACK_S : Bool := false;   // Request: acknowledge step at parameter S_NO
         REG_S : Bool := false;   // Request: register step indicated in S_NO
         T_PREV : Bool := false;   // Request: output previous valid transition in T_NO
         T_NEXT : Bool := false;   // Request: output next valid transition in T_NO
         LOCK : Bool := true;   // Status: interlocks activated
         SUP : Bool := true;   // Status: supervisions activated
         ACKREQ : Bool := true;   // Status: acknowledgment required
         SSKIP : Bool := false;   // Status: "Skip steps" enabled
         OFF : Bool := false;   // Request: deactivate all steps
         INIT : Bool := true;   // Request: set sequence to initial state
         HALT : Bool := false;   // Status: sequence halted
         TMS_HALT : Bool := false;   // Status: all internal timers held
         OPS_ZERO : Bool := false;   // Status: set all operands processed with N, L, D instructions to 0
         SACT_DISP : Bool := true;   // Status: display active steps only
         SEF_DISP : Bool := false;   // Status: display only steps with errors and disrupted steps
         SALL_DISP : Bool := false;   // Status: display all steps
         S_PREV : Bool := false;   // Request: output previous step to S_NO
         S_NEXT : Bool := false;   // Request: Output next step at S_NO parameter
         S_SELOK : Bool := false;   // Request: output step number from S_SEL to S_NO
         S_ON : Bool := false;   // Request: activate step indicated in S_NO
         S_OFF : Bool := false;   // Request: deactivate step at parameter S_NO
         T_PUSH : Bool := false;   // Request: transition switching enabled
         REG : Bool := false;   // Request: register all interlock and supervision errors
         ACK : Bool := false;   // Request: acknowledge all interlock and supervision errors
         IL_PERM : Bool := false;   // Status: permanent processing of all interlocks
         T_PERM : Bool := false;   // Status: permanent processing of all transitions
         ILP_MAN : Bool := false;   // Status: permanent processing of all interlocks in manual mode
      END_STRUCT;
      TICKS : Struct   // Clock speeds
         DELTA : Time := T#0ms;   // Time difference between cycles
         OLD : Time := T#0ms;   // 10 ms clock counter value in last cycle
         NEW : Time := T#0ms;   // 10 ms clock counter value in this cycle
      END_STRUCT;
      SQ_FLAGS : Struct   // Sequence bit memory
         ERR_FLT : Bool := false;   // Interlock and supervision group error
         ERROR : Bool := false;   // Interlock group error
         FAULT : Bool := false;   // Supervision group error
         RT_FAIL : Bool := false;   // Runtime error
         NO_SNO : Bool := false;   // Requested step number not found
         NF_OFL : Bool := false;   // Overflow: too many ON or OFF requests
         SA_OFL : Bool := false;   // Overflow: too many steps active
         TV_OFL : Bool := false;   // Overflow: too many valid transitions
         MSG_OFL : Bool := false;   // Overflow: not enough system resources for ALARM_S
         NO_SWI : Bool := false;   // Do not switch in this cycle
         CYC_OP : Bool := false;   // Cyclic execution of the sequence after initialization
         AS_MSG : Bool := true;   // Alarms during runtime enabled or disabled by instruction
         AS_SEND : Bool := false;   // Send alarms from WR_USMSG or only enter in diagnostics buffer
         SQ_BUSY : Bool := false;   // Internal edge bit memory for sequence processing
         SA_BUSY : Bool := false;   // Internal edge bit memory for sequence processing
         AS_SIG : Bool := false;   // Edge bit memory for alarms from Alarm_S and Alarm_SQ
      END_STRUCT;
      S_PTR : DWord := 16#B20;
      S_PTR2 : DWord := 16#0;
      S_PTR3 : DWord := 16#1E30;
      S_PTR4 : DWord := 16#1DA0;
      T_PTR : DWord := 16#1D10;
      C_AR2 : DWord := 16#0;
      M_FBDB : DWord := 16#40000;
      M_SNO : Word := 16#0;
      M_EVID : Word := 16#0;
      M_EVIL : C_Alarm_s;
      M_EVSV : C_Alarm_s;
      M_EV : DWord := 16#1C20;
      CRIT : Array[0..31] of Bool;
      S_START : Byte := 16#0;
      S_IDX : Byte := 16#0;
      S_INT : Int := 72;
      S_TMP : Byte := 16#0;
      T_START : Byte := 16#0;
      T_IDX : Byte := 16#0;
      T_TMP : Byte := 16#0;
      T_TMP2 : Byte := 16#00;
      TV_POT : Byte := 16#06;
      RETURN1 : Byte := 16#0;
      RETURN2 : Byte := 16#0;
      SINI : Array[0..2] of Byte;
      LSTT : Array[0..19] of Byte;
      ATAJ : Array[0..19] of Byte;
      ATAB : Array[0..19] of Byte;
      PSTT : Array[0..19] of Byte;
      NSTT : Array[0..19] of Byte;
      ASSJ : Array[0..15] of Byte;
      ASSB : Array[0..15] of Byte;
      PTTS : Array[0..15] of Byte;
      NTTS : Array[0..15] of Byte;
      PRE_CNT : Word := 16#1;
      POST_CNT : Word := 16#1;
      ADR_COND : Word := 16#0;
      MAX_TVAL : Byte := 16#6;
      MAX_SACT : Byte := 16#1;
      MAX_CRIT : Byte := 16#4;
      T_CNT : Byte := 16#13;
      SUP_CNT : Byte := 16#0;
      LOCK_CNT : Byte := 16#0;
      S_CNT : Byte := 16#F;
      SQ_CNT : Byte := 16#1;
      PRS_INPAR : DWord := 16#E000FEC8;
      PRS_OUTPAR : DWord := 16#E000800F;
      GC_FLAGS : Struct
         T_MACH : Byte := 16#EB;
         COND_ED : Byte := 16#E3;
         W_LEVEL : Byte := 16#D5;
         FB_IF : Byte := 16#FA;
         AS_MSG : Word := 16#404;
         SSB : Word := 16#108;
         DILG : Word := 16#500;
         ADDR_T0 : Word := 16#24;
         CRIT_AVAIL : Bool := false;
         SSKIP_AVAIL : Bool := true;
         SSKIP_ON : Bool := false;
         ACK_REQ : Bool := true;
         SYNC_AVAIL : Bool := true;
         ILP_MAN : Bool := false;
         SWM_LOCKED : Bool := false;
         SAVE_SW : Bool := true;
      END_STRUCT;
      G7_FBMARK : Byte := 16#3C;
      G7_RELEASE : Byte := 16#3C;
      G7_ID2 : Byte := 16#37;
      G7_ID1 : Byte := 16#47;
   END_VAR
   // SW_SQTS[0] := 16#6;
   // SW_SQTS[2] := 16#1;
   // SW_SQTS[3] := 16#1;
   // SW_SQTS[4] := 16#1;
   // SW_SQTS[5] := 16#1;
   // SW_SQTS[6] := 16#2;
   // TVX[0] := 16#1;
   // TTX[0] := 16#1;
   // TSX[0] := 16#1;
   // S00X[0] := 16#1;
   // SOFFX[0] := 16#1;
   // SONX[0] := 16#1;
   // SAX[0] := 16#1;
   // SERRX[0] := 16#1;
   // SMX[0] := 16#1;
   // S0X[0] := 16#1;
   // S1X[0] := 16#1;
   // SINI[0] := 16#2;
   // SINI[1] := 16#1;
   // SINI[2] := 0;
   // LSTT[0] := 0;
   // LSTT[1] := 0;
   // LSTT[2] := 0;
   // LSTT[3] := 0;
   // LSTT[4] := 0;
   // LSTT[5] := 16#1;
   // LSTT[6] := 0;
   // LSTT[7] := 16#1;
   // ATAJ[0] := 0;
   // ATAJ[1] := 16#1;
   // ATAJ[2] := 16#2;
   // ATAJ[3] := 16#3;
   // ATAJ[4] := 16#4;
   // ATAJ[5] := 16#5;
   // ATAJ[6] := 16#6;
   // ATAJ[7] := 16#7;
   // ATAB[0] := 0;
   // ATAB[1] := 16#6;
   // ATAB[2] := 16#2;
   // ATAB[3] := 16#3;
   // ATAB[4] := 16#4;
   // ATAB[5] := 16#5;
   // ATAB[6] := 16#8;
   // ATAB[7] := 16#7;
   // PSTT[0] := 0;
   // PSTT[1] := 16#1;
   // PSTT[2] := 16#2;
   // PSTT[3] := 16#3;
   // PSTT[4] := 16#4;
   // PSTT[5] := 16#5;
   // PSTT[6] := 16#1;
   // PSTT[7] := 16#6;
   // NSTT[0] := 16#1;
   // NSTT[1] := 16#2;
   // NSTT[2] := 16#3;
   // NSTT[3] := 16#4;
   // NSTT[4] := 16#5;
   // NSTT[5] := 16#1;
   // NSTT[6] := 16#6;
   // NSTT[7] := 16#1;
   // ASSJ[0] := 0;
   // ASSJ[1] := 16#1;
   // ASSJ[2] := 16#2;
   // ASSJ[3] := 16#3;
   // ASSJ[4] := 16#4;
   // ASSJ[5] := 16#5;
   // ASSJ[6] := 16#6;
   // ASSB[0] := 0;
   // ASSB[1] := 16#1;
   // ASSB[2] := 16#2;
   // ASSB[3] := 16#3;
   // ASSB[4] := 16#4;
   // ASSB[5] := 16#5;
   // ASSB[6] := 16#6;
   // PTTS[0] := 0;
   // PTTS[2] := 16#1;
   // PTTS[3] := 16#2;
   // PTTS[4] := 16#3;
   // PTTS[5] := 16#4;
   // PTTS[6] := 16#6;
   // NTTS[0] := 0;
   // NTTS[1] := 16#1;
   // NTTS[2] := 16#2;
   // NTTS[3] := 16#3;
   // NTTS[4] := 16#4;
   // NTTS[5] := 16#5;
   // NTTS[6] := 16#7;
   // SW_SQTS[7] := 16#3;
   // SW_SQTS[8] := 16#3;
   // SW_SQTS[9] := 16#3;
   // SW_SQTS[10] := 16#3;
   // SW_SQTS[11] := 16#4;
   // SW_SQTS[12] := 16#4;
   // SW_SQTS[13] := 16#4;
   // SW_SQTS[14] := 16#5;
   // SW_SQTS[15] := 16#5;
   // LSTT[8] := 0;
   // LSTT[9] := 0;
   // LSTT[10] := 0;
   // LSTT[11] := 0;
   // LSTT[12] := 16#1;
   // LSTT[13] := 0;
   // LSTT[14] := 0;
   // LSTT[15] := 0;
   // LSTT[16] := 16#1;
   // LSTT[17] := 0;
   // LSTT[18] := 0;
   // LSTT[19] := 16#1;
   // ATAJ[8] := 16#8;
   // ATAJ[9] := 16#9;
   // ATAJ[10] := 16#A;
   // ATAJ[11] := 16#B;
   // ATAJ[12] := 16#C;
   // ATAJ[13] := 16#D;
   // ATAJ[14] := 16#E;
   // ATAJ[15] := 16#F;
   // ATAJ[16] := 16#10;
   // ATAJ[17] := 16#11;
   // ATAJ[18] := 16#12;
   // ATAJ[19] := 16#13;
   // ATAB[8] := 16#D;
   // ATAB[9] := 16#9;
   // ATAB[10] := 16#A;
   // ATAB[11] := 16#B;
   // ATAB[12] := 16#C;
   // ATAB[13] := 16#11;
   // ATAB[14] := 16#E;
   // ATAB[15] := 16#F;
   // ATAB[16] := 16#10;
   // ATAB[17] := 16#1;
   // ATAB[18] := 16#12;
   // ATAB[19] := 16#13;
   // PSTT[8] := 16#1;
   // PSTT[9] := 16#7;
   // PSTT[10] := 16#8;
   // PSTT[11] := 16#9;
   // PSTT[12] := 16#A;
   // PSTT[13] := 16#1;
   // PSTT[14] := 16#B;
   // PSTT[15] := 16#C;
   // PSTT[16] := 16#D;
   // PSTT[17] := 16#1;
   // PSTT[18] := 16#E;
   // PSTT[19] := 16#F;
   // NSTT[8] := 16#7;
   // NSTT[9] := 16#8;
   // NSTT[10] := 16#9;
   // NSTT[11] := 16#A;
   // NSTT[12] := 16#1;
   // NSTT[13] := 16#B;
   // NSTT[14] := 16#C;
   // NSTT[15] := 16#D;
   // NSTT[16] := 16#1;
   // NSTT[17] := 16#E;
   // NSTT[18] := 16#F;
   // NSTT[19] := 16#1;
   // ASSJ[7] := 16#7;
   // ASSJ[8] := 16#8;
   // ASSJ[9] := 16#9;
   // ASSJ[10] := 16#A;
   // ASSJ[11] := 16#B;
   // ASSJ[12] := 16#C;
   // ASSJ[13] := 16#D;
   // ASSJ[14] := 16#E;
   // ASSJ[15] := 16#F;
   // ASSB[7] := 16#7;
   // ASSB[8] := 16#8;
   // ASSB[9] := 16#9;
   // ASSB[10] := 16#A;
   // ASSB[11] := 16#B;
   // ASSB[12] := 16#C;
   // ASSB[13] := 16#D;
   // ASSB[14] := 16#E;
   // ASSB[15] := 16#F;
   // PTTS[7] := 16#8;
   // PTTS[8] := 16#9;
   // PTTS[9] := 16#A;
   // PTTS[10] := 16#B;
   // PTTS[11] := 16#D;
   // PTTS[12] := 16#E;
   // PTTS[13] := 16#F;
   // PTTS[14] := 16#11;
   // PTTS[15] := 16#12;
   // NTTS[7] := 16#9;
   // NTTS[8] := 16#A;
   // NTTS[9] := 16#B;
   // NTTS[10] := 16#C;
   // NTTS[11] := 16#E;
   // NTTS[12] := 16#F;
   // NTTS[13] := 16#10;
   // NTTS[14] := 16#12;
   // NTTS[15] := 16#13;
BEGIN
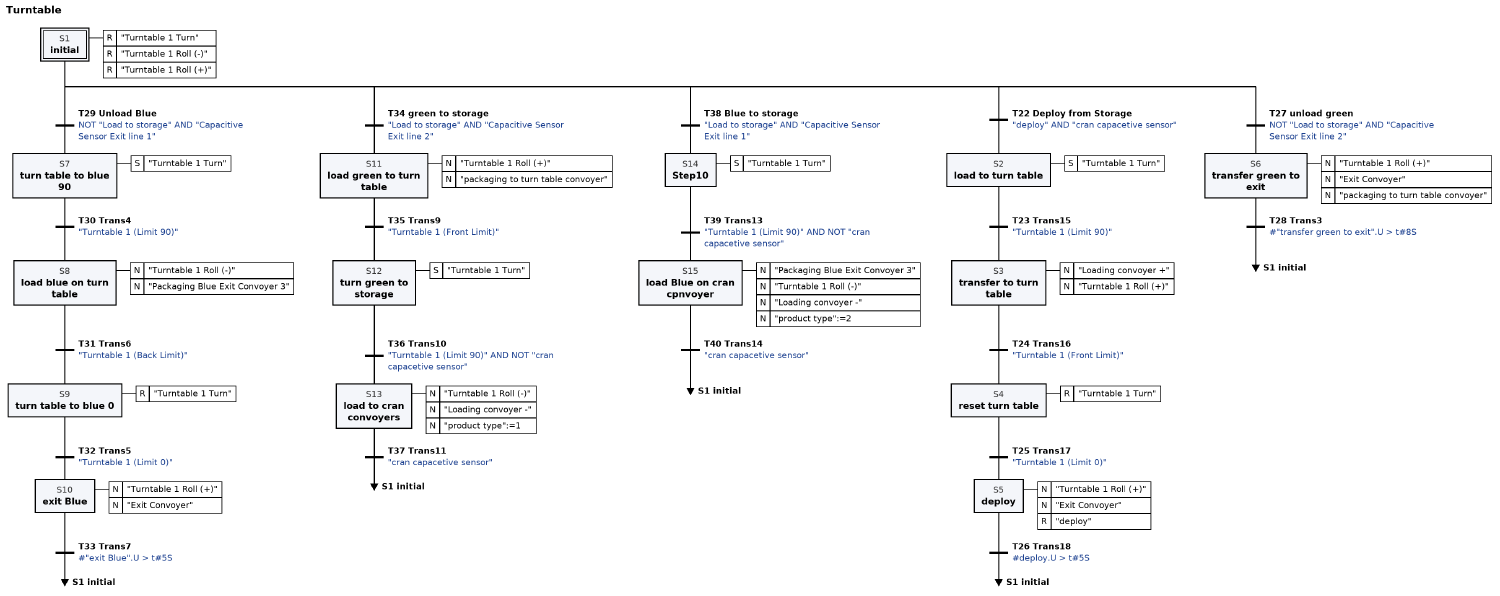
   // sequencer 1
   INITIAL_STEP initial:   // S1
              R    "Turntable 1 Turn"
              R    "Turntable 1 Roll (-)"
              R    "Turntable 1 Roll (+)"
   END_STEP
   TRANSITION "Unload Blue" FROM initial TO "turn table to blue 90"   // T29
      := NOT "Load to storage" AND "Capacitive Sensor Exit line 1";
   END_TRANSITION
   TRANSITION "green to storage" FROM initial TO "load green to turn table"   // T34
      := "Load to storage" AND "Capacitive Sensor Exit line 2";
   END_TRANSITION
   TRANSITION "Blue to storage" FROM initial TO Step10   // T38
      := "Load to storage" AND "Capacitive Sensor Exit line 1";
   END_TRANSITION
   TRANSITION "Deploy from Storage" FROM initial TO "load to turn table"   // T22
      := "deploy" AND "cran capacetive sensor";
   END_TRANSITION
   TRANSITION "unload green" FROM initial TO "transfer green to exit"   // T27
      := NOT "Load to storage" AND "Capacitive Sensor Exit line 2";
   END_TRANSITION
   STEP "reset turn table":   // S4
              R    "Turntable 1 Turn"
   END_STEP
   TRANSITION Trans17 FROM "reset turn table" TO deploy   // T25
      := "Turntable 1 (Limit 0)";
   END_TRANSITION
   STEP "turn table to blue 90":   // S7
              S    "Turntable 1 Turn"
   END_STEP
   TRANSITION Trans4 FROM "turn table to blue 90" TO "load blue on turn table"   // T30
      := "Turntable 1 (Limit 90)";
   END_TRANSITION
   STEP "turn table to blue 0":   // S9
              R    "Turntable 1 Turn"
   END_STEP
   TRANSITION Trans5 FROM "turn table to blue 0" TO "exit Blue"   // T32
      := "Turntable 1 (Limit 0)";
   END_TRANSITION
   STEP "load blue on turn table":   // S8
              N    "Turntable 1 Roll (-)"
              N    "Packaging Blue Exit Convoyer 3"
   END_STEP
   TRANSITION Trans6 FROM "load blue on turn table" TO "turn table to blue 0"   // T31
      := "Turntable 1 (Back Limit)";
   END_TRANSITION
   STEP "exit Blue":   // S10
              N    "Turntable 1 Roll (+)"
              N    "Exit Convoyer"
   END_STEP
   TRANSITION Trans7 FROM "exit Blue" TO initial   // T33, jump
      := #"exit Blue".U > t#5S;
   END_TRANSITION
   STEP "load green to turn table":   // S11
              N    "Turntable 1 Roll (+)"
              N    "packaging to turn table convoyer"
   END_STEP
   TRANSITION Trans9 FROM "load green to turn table" TO "turn green to storage"   // T35
      := "Turntable 1 (Front Limit)";
   END_TRANSITION
   STEP "turn green to storage":   // S12
              S    "Turntable 1 Turn"
   END_STEP
   TRANSITION Trans10 FROM "turn green to storage" TO "load to cran convoyers"   // T36
      := "Turntable 1 (Limit 90)" AND NOT "cran capacetive sensor";
   END_TRANSITION
   STEP "load to cran convoyers":   // S13
              N    "Turntable 1 Roll (-)"
              N    "Loading convoyer -"
              N    "product type":=1
   END_STEP
   TRANSITION Trans11 FROM "load to cran convoyers" TO initial   // T37, jump
      := "cran capacetive sensor";
   END_TRANSITION
   STEP Step10:   // S14
              S    "Turntable 1 Turn"
   END_STEP
   TRANSITION Trans13 FROM Step10 TO "load Blue on cran cpnvoyer"   // T39
      := "Turntable 1 (Limit 90)" AND NOT "cran capacetive sensor";
   END_TRANSITION
   STEP "load Blue on cran cpnvoyer":   // S15
              N    "Packaging Blue Exit Convoyer 3"
              N    "Turntable 1 Roll (-)"
              N    "Loading convoyer -"
              N    "product type":=2
   END_STEP
   TRANSITION Trans14 FROM "load Blue on cran cpnvoyer" TO initial   // T40, jump
      := "cran capacetive sensor";
   END_TRANSITION
   STEP "load to turn table":   // S2
              S    "Turntable 1 Turn"
   END_STEP
   TRANSITION Trans15 FROM "load to turn table" TO "transfer to turn table"   // T23
      := "Turntable 1 (Limit 90)";
   END_TRANSITION
   STEP "transfer to turn table":   // S3
              N    "Loading convoyer +"
              N    "Turntable 1 Roll (+)"
   END_STEP
   TRANSITION Trans16 FROM "transfer to turn table" TO "reset turn table"   // T24
      := "Turntable 1 (Front Limit)";
   END_TRANSITION
   STEP "transfer green to exit":   // S6
              N    "Turntable 1 Roll (+)"
              N    "Exit Convoyer"
              N    "packaging to turn table convoyer"
   END_STEP
   TRANSITION Trans3 FROM "transfer green to exit" TO initial   // T28, jump
      := #"transfer green to exit".U > t#8S;
   END_TRANSITION
   STEP deploy:   // S5
              N    "Turntable 1 Roll (+)"
              N    "Exit Convoyer"
              R    "deploy"
   END_STEP
   TRANSITION Trans18 FROM deploy TO initial   // T26, jump
      := #deploy.U > t#5S;
   END_TRANSITION
END_FUNCTION_BLOCK

FUNCTION_BLOCK "stacker"   // FB5, GRAPH
{ S7_Optimized_Access := 'FALSE' }
VERSION : 0.1
   VAR_INPUT
      OFF_SQ : Bool := false;   // Turn sequence off
      INIT_SQ : Bool := false;   // Set sequence to initial state
      ACK_EF : Bool := false;   // Acknowledge all errors and faults
      S_PREV : Bool := false;   // Output previous step in parameter S_NO
      S_NEXT : Bool := false;   // Indicate next step in parameter S_NO
      SW_AUTO : Bool := false;   // Automatic mode
      SW_TAP : Bool := false;   // Semiautomatic/switch with transition
      SW_TOP : Bool := false;   // Semiautomatic/ignore transition
      SW_MAN : Bool := false;   // Manual mode
      S_SEL : Int := 0;   // Select step to be output to S_NO
      S_ON : Bool := false;   // Activate step indicated in S_NO
      S_OFF : Bool := false;   // Deactivate step indicated S_NO
      T_PUSH : Bool := false;   // Enable transition to switch in semi automatic mode
   END_VAR
   VAR_OUTPUT
      S_NO : Int := 0;   // Step number
      S_MORE : Bool := false;   // More steps are available and can be shown in S_NO
      S_ACTIVE : Bool := false;   // Step indicated in S_NO is active
      ERR_FLT : Bool := false;   // Interlock or supervision group error
      AUTO_ON : Bool := false;   // Automatic mode is active
      TAP_ON : Bool := false;   // Semiautomatic mode/step with transition enabled
      TOP_ON : Bool := false;   // Semiautomatic mode/ignore transition enabled
      MAN_ON : Bool := false;   // Manual mode is active
   END_VAR
   VAR
      SWITCH : Array[0..0] of DWord;
      SW_SQTS : Array[0..19] of Byte;
      SW_ADDR : Word := 16#A;
      G7T_0 : GraphTransition;
      G7S_0 : GraphStep;
      PRE_CRIT : Array[0..0] of DWord;
      POST_CRIT : Array[0..0] of DWord;
      TVX : Array[0..4] of Byte;
      TTX : Array[0..4] of Byte;
      TSX : Array[0..2] of Byte;
      S00X : Array[0..2] of Byte;
      SOFFX : Array[0..2] of Byte;
      SONX : Array[0..2] of Byte;
      SAX : Array[0..2] of Byte;
      SERRX : Array[0..20] of Byte;
      SMX : Array[0..20] of Byte;
      S0X : Array[0..20] of Byte;
      S1X : Array[0..20] of Byte;
      S_DISPLAY : Int;   // Internal display of output parameter S_NO
      S_SEL_OLD : Int;   // Previous value in S_SEL
      S_DISPIDX : Byte;   // Index of the step in S_NO
      T_DISPIDX : Byte;   // Index of the transition displayed in T_NO
      MOPEDGE : Struct
         AUTO : Bool := false;
         MAN : Bool := false;
         TAP : Bool := false;
         TOP : Bool := false;
         ACK_S : Bool := false;
         REG_S : Bool := false;
         T_PREV : Bool := false;
         T_NEXT : Bool := false;
         LOCK : Bool := false;
         SUP : Bool := false;
         ACKREQ : Bool := false;
         SSKIP : Bool := false;
         OFF : Bool := false;
         INIT : Bool := false;
         HALT : Bool := false;
         TMS_HALT : Bool := false;
         OPS_ZERO : Bool := false;
         SACT_DISP : Bool := false;
         SEF_DISP : Bool := false;
         SALL_DISP : Bool := false;
         S_PREV : Bool := false;
         S_NEXT : Bool := false;
         S_SELOK : Bool := false;
         S_ON : Bool := false;
         S_OFF : Bool := false;
         T_PUSH : Bool := false;
         REG : Bool := false;
         ACK : Bool := false;
         IL_PERM : Bool := false;
         T_PERM : Bool := false;
         ILP_MAN : Bool := false;
      END_STRUCT;
      MOP : Struct   // Mode
         AUTO : Bool := true;   // Status: automatic mode
         MAN : Bool := false;   // Status: manual mode
         TAP : Bool := false;   // Status: semi automatic/switch with transition
         TOP : Bool := false;   // Status: semi automatic/ignore transition
         ACK_S : Bool := false;   // Request: acknowledge step at parameter S_NO
         REG_S : Bool := false;   // Request: register step indicated in S_NO
         T_PREV : Bool := false;   // Request: output previous valid transition in T_NO
         T_NEXT : Bool := false;   // Request: output next valid transition in T_NO
         LOCK : Bool := true;   // Status: interlocks activated
         SUP : Bool := true;   // Status: supervisions activated
         ACKREQ : Bool := true;   // Status: acknowledgment required
         SSKIP : Bool := false;   // Status: "Skip steps" enabled
         OFF : Bool := false;   // Request: deactivate all steps
         INIT : Bool := true;   // Request: set sequence to initial state
         HALT : Bool := false;   // Status: sequence halted
         TMS_HALT : Bool := false;   // Status: all internal timers held
         OPS_ZERO : Bool := false;   // Status: set all operands processed with N, L, D instructions to 0
         SACT_DISP : Bool := true;   // Status: display active steps only
         SEF_DISP : Bool := false;   // Status: display only steps with errors and disrupted steps
         SALL_DISP : Bool := false;   // Status: display all steps
         S_PREV : Bool := false;   // Request: output previous step to S_NO
         S_NEXT : Bool := false;   // Request: Output next step at S_NO parameter
         S_SELOK : Bool := false;   // Request: output step number from S_SEL to S_NO
         S_ON : Bool := false;   // Request: activate step indicated in S_NO
         S_OFF : Bool := false;   // Request: deactivate step at parameter S_NO
         T_PUSH : Bool := false;   // Request: transition switching enabled
         REG : Bool := false;   // Request: register all interlock and supervision errors
         ACK : Bool := false;   // Request: acknowledge all interlock and supervision errors
         IL_PERM : Bool := false;   // Status: permanent processing of all interlocks
         T_PERM : Bool := false;   // Status: permanent processing of all transitions
         ILP_MAN : Bool := false;   // Status: permanent processing of all interlocks in manual mode
      END_STRUCT;
      TICKS : Struct   // Clock speeds
         DELTA : Time := T#0ms;   // Time difference between cycles
         OLD : Time := T#0ms;   // 10 ms clock counter value in last cycle
         NEW : Time := T#0ms;   // 10 ms clock counter value in this cycle
      END_STRUCT;
      SQ_FLAGS : Struct   // Sequence bit memory
         ERR_FLT : Bool := false;   // Interlock and supervision group error
         ERROR : Bool := false;   // Interlock group error
         FAULT : Bool := false;   // Supervision group error
         RT_FAIL : Bool := false;   // Runtime error
         NO_SNO : Bool := false;   // Requested step number not found
         NF_OFL : Bool := false;   // Overflow: too many ON or OFF requests
         SA_OFL : Bool := false;   // Overflow: too many steps active
         TV_OFL : Bool := false;   // Overflow: too many valid transitions
         MSG_OFL : Bool := false;   // Overflow: not enough system resources for ALARM_S
         NO_SWI : Bool := false;   // Do not switch in this cycle
         CYC_OP : Bool := false;   // Cyclic execution of the sequence after initialization
         AS_MSG : Bool := true;   // Alarms during runtime enabled or disabled by instruction
         AS_SEND : Bool := false;   // Send alarms from WR_USMSG or only enter in diagnostics buffer
         SQ_BUSY : Bool := false;   // Internal edge bit memory for sequence processing
         SA_BUSY : Bool := false;   // Internal edge bit memory for sequence processing
         AS_SIG : Bool := false;   // Edge bit memory for alarms from Alarm_S and Alarm_SQ
      END_STRUCT;
      S_PTR : DWord := 16#BA0;
      S_PTR2 : DWord := 16#0;
      S_PTR3 : DWord := 16#22F0;
      S_PTR4 : DWord := 16#2240;
      T_PTR : DWord := 16#2190;
      C_AR2 : DWord := 16#0;
      M_FBDB : DWord := 16#50000;
      M_SNO : Word := 16#0;
      M_EVID : Word := 16#0;
      M_EVIL : C_Alarm_s;
      M_EVSV : C_Alarm_s;
      M_EV : DWord := 16#2080;
      CRIT : Array[0..31] of Bool;
      S_START : Byte := 16#0;
      S_IDX : Byte := 16#0;
      S_INT : Int := 72;
      S_TMP : Byte := 16#0;
      T_START : Byte := 16#0;
      T_IDX : Byte := 16#0;
      T_TMP : Byte := 16#0;
      T_TMP2 : Byte := 16#00;
      TV_POT : Byte := 16#06;
      RETURN1 : Byte := 16#0;
      RETURN2 : Byte := 16#0;
      SINI : Array[0..2] of Byte;
      LSTT : Array[0..20] of Byte;
      ATAJ : Array[0..20] of Byte;
      ATAB : Array[0..20] of Byte;
      PSTT : Array[0..20] of Byte;
      NSTT : Array[0..20] of Byte;
      ASSJ : Array[0..19] of Byte;
      ASSB : Array[0..19] of Byte;
      PTTS : Array[0..19] of Byte;
      NTTS : Array[0..19] of Byte;
      PRE_CNT : Word := 16#1;
      POST_CNT : Word := 16#1;
      ADR_COND : Word := 16#0;
      MAX_TVAL : Byte := 16#3;
      MAX_SACT : Byte := 16#1;
      MAX_CRIT : Byte := 16#4;
      T_CNT : Byte := 16#14;
      SUP_CNT : Byte := 16#0;
      LOCK_CNT : Byte := 16#0;
      S_CNT : Byte := 16#13;
      SQ_CNT : Byte := 16#1;
      PRS_INPAR : DWord := 16#E000FEC8;
      PRS_OUTPAR : DWord := 16#E000800F;
      GC_FLAGS : Struct
         T_MACH : Byte := 16#EB;
         COND_ED : Byte := 16#E3;
         W_LEVEL : Byte := 16#D5;
         FB_IF : Byte := 16#FA;
         AS_MSG : Word := 16#404;
         SSB : Word := 16#108;
         DILG : Word := 16#5B6;
         ADDR_T0 : Word := 16#24;
         CRIT_AVAIL : Bool := false;
         SSKIP_AVAIL : Bool := true;
         SSKIP_ON : Bool := false;
         ACK_REQ : Bool := true;
         SYNC_AVAIL : Bool := true;
         ILP_MAN : Bool := false;
         SWM_LOCKED : Bool := false;
         SAVE_SW : Bool := true;
      END_STRUCT;
      G7_FBMARK : Byte := 16#3C;
      G7_RELEASE : Byte := 16#3C;
      G7_ID2 : Byte := 16#37;
      G7_ID1 : Byte := 16#47;
   END_VAR
   // SW_SQTS[0] := 16#3;
   // TVX[0] := 16#1;
   // TTX[0] := 16#1;
   // TSX[0] := 16#1;
   // S00X[0] := 16#1;
   // SOFFX[0] := 16#1;
   // SONX[0] := 16#1;
   // SAX[0] := 16#1;
   // SERRX[0] := 16#1;
   // SMX[0] := 16#1;
   // S0X[0] := 16#1;
   // S1X[0] := 16#1;
   // SINI[0] := 16#2;
   // SINI[1] := 16#1;
   // SINI[2] := 0;
   // LSTT[0] := 0;
   // LSTT[1] := 0;
   // LSTT[2] := 0;
   // LSTT[3] := 0;
   // LSTT[4] := 0;
   // LSTT[5] := 0;
   // LSTT[6] := 0;
   // ATAJ[0] := 0;
   // ATAJ[1] := 16#1;
   // ATAJ[2] := 16#2;
   // ATAJ[3] := 16#3;
   // ATAJ[4] := 16#4;
   // ATAJ[5] := 16#5;
   // ATAJ[6] := 16#6;
   // ATAB[0] := 0;
   // ATAB[1] := 16#B;
   // ATAB[2] := 16#2;
   // ATAB[3] := 16#3;
   // ATAB[4] := 16#4;
   // ATAB[5] := 16#5;
   // ATAB[6] := 16#6;
   // PSTT[0] := 0;
   // PSTT[1] := 16#5;
   // PSTT[2] := 16#2;
   // PSTT[3] := 16#3;
   // PSTT[4] := 16#4;
   // PSTT[5] := 16#1;
   // PSTT[6] := 16#6;
   // NSTT[0] := 16#1;
   // NSTT[1] := 16#2;
   // NSTT[2] := 16#3;
   // NSTT[3] := 16#4;
   // NSTT[4] := 16#6;
   // NSTT[5] := 16#5;
   // ASSJ[0] := 0;
   // ASSJ[1] := 16#1;
   // ASSJ[2] := 16#2;
   // ASSJ[3] := 16#3;
   // ASSJ[4] := 16#4;
   // ASSJ[5] := 16#5;
   // ASSJ[6] := 16#6;
   // ASSB[0] := 0;
   // ASSB[1] := 16#1;
   // ASSB[2] := 16#2;
   // ASSB[3] := 16#3;
   // ASSB[4] := 16#4;
   // ASSB[5] := 16#5;
   // ASSB[6] := 16#6;
   // PTTS[0] := 0;
   // PTTS[2] := 16#1;
   // PTTS[3] := 16#2;
   // PTTS[4] := 16#3;
   // PTTS[5] := 16#5;
   // PTTS[6] := 16#4;
   // NTTS[0] := 0;
   // NTTS[1] := 16#5;
   // NTTS[2] := 16#2;
   // NTTS[3] := 16#3;
   // NTTS[4] := 16#4;
   // NTTS[5] := 16#1;
   // NTTS[6] := 16#6;
   // LSTT[7] := 0;
   // ATAJ[7] := 16#7;
   // ATAB[7] := 16#7;
   // PSTT[7] := 16#7;
   // NSTT[6] := 16#7;
   // ASSJ[7] := 16#7;
   // ASSB[7] := 16#7;
   // PTTS[7] := 16#6;
   // NTTS[7] := 16#7;
   // LSTT[8] := 0;
   // LSTT[9] := 0;
   // LSTT[10] := 0;
   // ATAJ[8] := 16#8;
   // ATAJ[9] := 16#9;
   // ATAJ[10] := 16#A;
   // ATAB[8] := 16#8;
   // ATAB[9] := 16#9;
   // ATAB[10] := 16#A;
   // PSTT[8] := 16#8;
   // PSTT[9] := 16#9;
   // PSTT[10] := 16#A;
   // NSTT[7] := 16#8;
   // NSTT[8] := 16#9;
   // NSTT[9] := 16#A;
   // NSTT[10] := 16#B;
   // ASSJ[8] := 16#8;
   // ASSJ[9] := 16#9;
   // ASSJ[10] := 16#A;
   // ASSB[8] := 16#8;
   // ASSB[9] := 16#9;
   // ASSB[10] := 16#A;
   // PTTS[8] := 16#7;
   // PTTS[9] := 16#8;
   // PTTS[10] := 16#9;
   // NTTS[8] := 16#8;
   // NTTS[9] := 16#9;
   // NTTS[10] := 16#A;
   // SW_SQTS[2] := 16#1;
   // SW_SQTS[3] := 16#1;
   // SW_SQTS[4] := 16#1;
   // SW_SQTS[6] := 16#1;
   // SW_SQTS[7] := 16#1;
   // SW_SQTS[8] := 16#1;
   // SW_SQTS[9] := 16#1;
   // SW_SQTS[10] := 16#1;
   // SW_SQTS[11] := 16#1;
   // SW_SQTS[12] := 16#2;
   // SW_SQTS[13] := 16#2;
   // SW_SQTS[14] := 16#2;
   // SW_SQTS[15] := 16#2;
   // SW_SQTS[16] := 16#2;
   // SW_SQTS[17] := 16#2;
   // SW_SQTS[18] := 16#2;
   // SW_SQTS[19] := 16#2;
   // LSTT[11] := 0;
   // LSTT[12] := 16#1;
   // LSTT[13] := 0;
   // LSTT[14] := 0;
   // LSTT[15] := 0;
   // LSTT[16] := 0;
   // LSTT[17] := 0;
   // LSTT[18] := 0;
   // LSTT[19] := 0;
   // LSTT[20] := 16#1;
   // ATAJ[11] := 16#B;
   // ATAJ[12] := 16#C;
   // ATAJ[13] := 16#D;
   // ATAJ[14] := 16#E;
   // ATAJ[15] := 16#F;
   // ATAJ[16] := 16#10;
   // ATAJ[17] := 16#11;
   // ATAJ[18] := 16#12;
   // ATAJ[19] := 16#13;
   // ATAJ[20] := 16#14;
   // ATAB[11] := 16#1;
   // ATAB[12] := 16#C;
   // ATAB[13] := 16#D;
   // ATAB[14] := 16#E;
   // ATAB[15] := 16#F;
   // ATAB[16] := 16#10;
   // ATAB[17] := 16#11;
   // ATAB[18] := 16#12;
   // ATAB[19] := 16#13;
   // ATAB[20] := 16#14;
   // PSTT[11] := 16#5;
   // PSTT[12] := 16#B;
   // PSTT[13] := 16#C;
   // PSTT[14] := 16#D;
   // PSTT[15] := 16#E;
   // PSTT[16] := 16#F;
   // PSTT[17] := 16#10;
   // PSTT[18] := 16#11;
   // PSTT[19] := 16#12;
   // PSTT[20] := 16#13;
   // NSTT[11] := 16#C;
   // NSTT[12] := 16#1;
   // NSTT[13] := 16#D;
   // NSTT[14] := 16#E;
   // NSTT[15] := 16#F;
   // NSTT[16] := 16#10;
   // NSTT[17] := 16#11;
   // NSTT[18] := 16#12;
   // NSTT[19] := 16#13;
   // NSTT[20] := 16#1;
   // ASSJ[11] := 16#B;
   // ASSJ[12] := 16#C;
   // ASSJ[13] := 16#D;
   // ASSJ[14] := 16#E;
   // ASSJ[15] := 16#F;
   // ASSJ[16] := 16#10;
   // ASSJ[17] := 16#11;
   // ASSJ[18] := 16#12;
   // ASSJ[19] := 16#13;
   // ASSB[11] := 16#B;
   // ASSB[12] := 16#C;
   // ASSB[13] := 16#D;
   // ASSB[14] := 16#E;
   // ASSB[15] := 16#F;
   // ASSB[16] := 16#10;
   // ASSB[17] := 16#11;
   // ASSB[18] := 16#12;
   // ASSB[19] := 16#13;
   // PTTS[11] := 16#A;
   // PTTS[12] := 16#B;
   // PTTS[13] := 16#D;
   // PTTS[14] := 16#E;
   // PTTS[15] := 16#F;
   // PTTS[16] := 16#10;
   // PTTS[17] := 16#11;
   // PTTS[18] := 16#12;
   // PTTS[19] := 16#13;
   // NTTS[11] := 16#C;
   // NTTS[12] := 16#D;
   // NTTS[13] := 16#E;
   // NTTS[14] := 16#F;
   // NTTS[15] := 16#10;
   // NTTS[16] := 16#11;
   // NTTS[17] := 16#12;
   // NTTS[18] := 16#13;
   // NTTS[19] := 16#14;
BEGIN
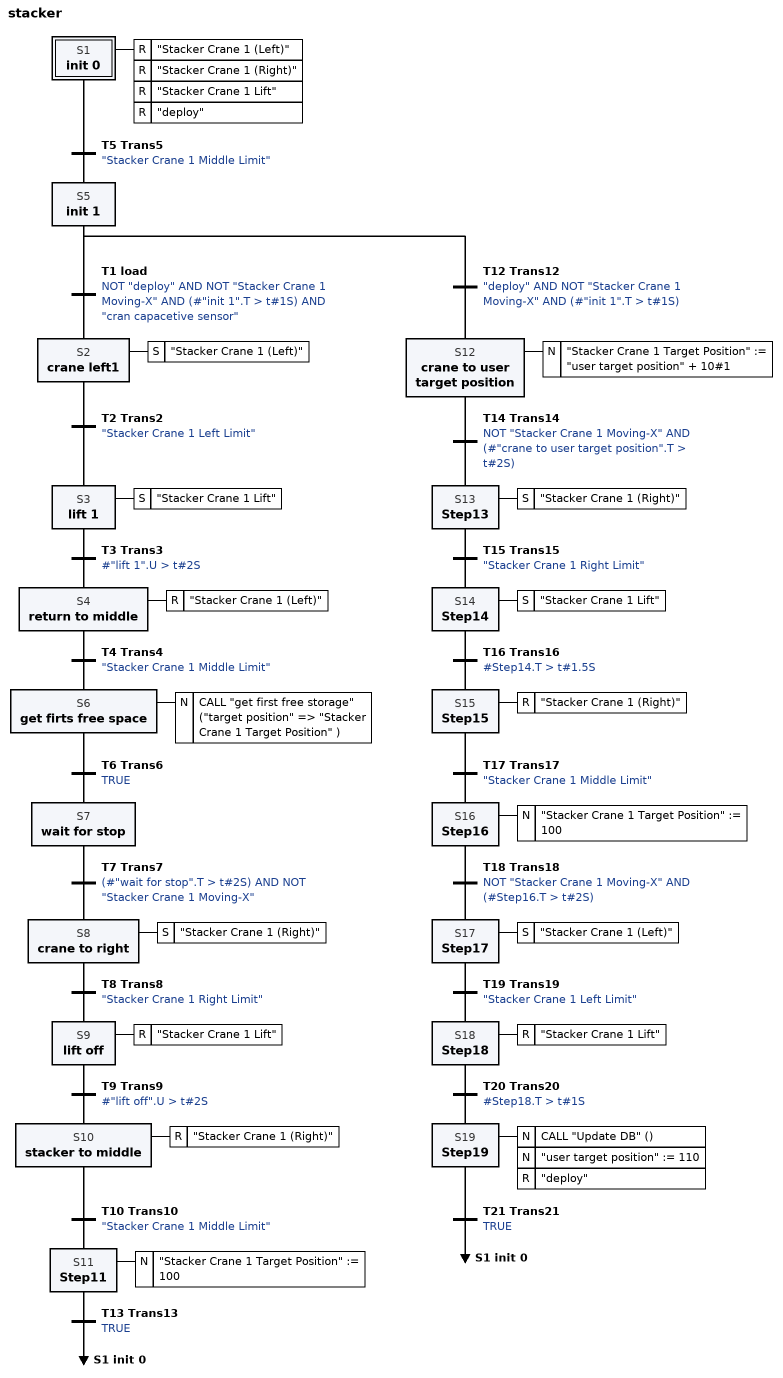
   // sequencer 1
   INITIAL_STEP "init 0":   // S1
              R    "Stacker Crane 1 (Left)"
              R    "Stacker Crane 1 (Right)"
              R    "Stacker Crane 1 Lift"
              R    "deploy"
   END_STEP
   TRANSITION Trans5 FROM "init 0" TO "init 1"   // T5
      := "Stacker Crane 1 Middle Limit";
   END_TRANSITION
   STEP "crane left1":   // S2
              S    "Stacker Crane 1 (Left)"
   END_STEP
   TRANSITION Trans2 FROM "crane left1" TO "lift 1"   // T2
      := "Stacker Crane 1 Left Limit";
   END_TRANSITION
   STEP "lift 1":   // S3
              S    "Stacker Crane 1 Lift"
   END_STEP
   TRANSITION Trans3 FROM "lift 1" TO "return to middle"   // T3
      := #"lift 1".U > t#2S;
   END_TRANSITION
   STEP "return to middle":   // S4
              R    "Stacker Crane 1 (Left)"
   END_STEP
   TRANSITION Trans4 FROM "return to middle" TO "get firts free space"   // T4
      := "Stacker Crane 1 Middle Limit";
   END_TRANSITION
   STEP "init 1":   // S5
   END_STEP
   TRANSITION load FROM "init 1" TO "crane left1"   // T1
      := NOT "deploy" AND NOT "Stacker Crane 1 Moving-X" AND (#"init 1".T > t#1S) AND "cran capacetive sensor";
   END_TRANSITION
   TRANSITION Trans12 FROM "init 1" TO "crane to user target position"   // T12
      := "deploy" AND NOT "Stacker Crane 1 Moving-X" AND (#"init 1".T > t#1S);
   END_TRANSITION
   STEP "get firts free space":   // S6
              N    CALL "get first free storage"
                   ("target position" => "Stacker Crane 1 Target Position"
                   )
   END_STEP
   TRANSITION Trans6 FROM "get firts free space" TO "wait for stop"   // T6
      := TRUE;
   END_TRANSITION
   STEP "wait for stop":   // S7
   END_STEP
   TRANSITION Trans7 FROM "wait for stop" TO "crane to right"   // T7
      := (#"wait for stop".T > t#2S) AND NOT "Stacker Crane 1 Moving-X";
   END_TRANSITION
   STEP "crane to right":   // S8
              S    "Stacker Crane 1 (Right)"
   END_STEP
   TRANSITION Trans8 FROM "crane to right" TO "lift off"   // T8
      := "Stacker Crane 1 Right Limit";
   END_TRANSITION
   STEP "lift off":   // S9
              R    "Stacker Crane 1 Lift"
   END_STEP
   TRANSITION Trans9 FROM "lift off" TO "stacker to middle"   // T9
      := #"lift off".U > t#2S;
   END_TRANSITION
   STEP "stacker to middle":   // S10
              R    "Stacker Crane 1 (Right)"
   END_STEP
   TRANSITION Trans10 FROM "stacker to middle" TO Step11   // T10
      := "Stacker Crane 1 Middle Limit";
   END_TRANSITION
   STEP Step11:   // S11
              N    "Stacker Crane 1 Target Position" := 100
   END_STEP
   TRANSITION Trans13 FROM Step11 TO "init 0"   // T13, jump
      := TRUE;
   END_TRANSITION
   STEP "crane to user target position":   // S12
              N    "Stacker Crane 1 Target Position" := "user target position" + 10#1
   END_STEP
   TRANSITION Trans14 FROM "crane to user target position" TO Step13   // T14
      := NOT "Stacker Crane 1 Moving-X" AND (#"crane to user target position".T > t#2S);
   END_TRANSITION
   STEP Step13:   // S13
              S    "Stacker Crane 1 (Right)"
   END_STEP
   TRANSITION Trans15 FROM Step13 TO Step14   // T15
      := "Stacker Crane 1 Right Limit";
   END_TRANSITION
   STEP Step14:   // S14
              S    "Stacker Crane 1 Lift"
   END_STEP
   TRANSITION Trans16 FROM Step14 TO Step15   // T16
      := #Step14.T > t#1.5S;
   END_TRANSITION
   STEP Step15:   // S15
              R    "Stacker Crane 1 (Right)"
   END_STEP
   TRANSITION Trans17 FROM Step15 TO Step16   // T17
      := "Stacker Crane 1 Middle Limit";
   END_TRANSITION
   STEP Step16:   // S16
              N    "Stacker Crane 1 Target Position" := 100
   END_STEP
   TRANSITION Trans18 FROM Step16 TO Step17   // T18
      := NOT "Stacker Crane 1 Moving-X" AND (#Step16.T > t#2S);
   END_TRANSITION
   STEP Step17:   // S17
              S    "Stacker Crane 1 (Left)"
   END_STEP
   TRANSITION Trans19 FROM Step17 TO Step18   // T19
      := "Stacker Crane 1 Left Limit";
   END_TRANSITION
   STEP Step18:   // S18
              R    "Stacker Crane 1 Lift"
   END_STEP
   TRANSITION Trans20 FROM Step18 TO Step19   // T20
      := #Step18.T > t#1S;
   END_TRANSITION
   STEP Step19:   // S19
              N    CALL "Update DB" ()
              N    "user target position" := 110
              R    "deploy"
   END_STEP
   TRANSITION Trans21 FROM Step19 TO "init 0"   // T21, jump
      := TRUE;
   END_TRANSITION
END_FUNCTION_BLOCK

FUNCTION "Storage system" : Void   // FC10, LAD
{ S7_Optimized_Access := 'FALSE' }
VERSION : 0.1
BEGIN

REGION Network 1
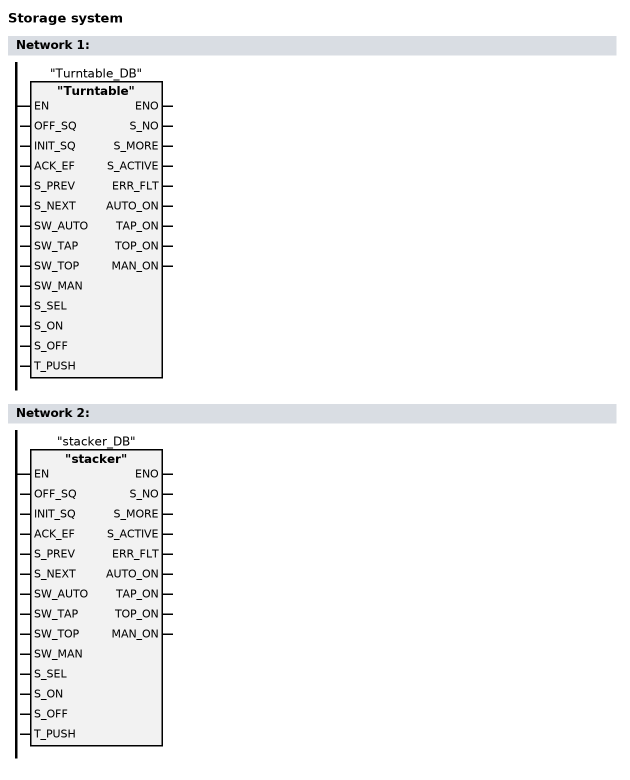
   RUNG wire#powerrail
      "Turntable_DB"(OFF_SQ :=, INIT_SQ :=, ACK_EF :=, S_PREV :=, S_NEXT :=, SW_AUTO :=, SW_TAP :=, SW_TOP :=, SW_MAN :=, S_SEL :=, S_ON :=, S_OFF :=, T_PUSH :=, S_NO =>, S_MORE =>, S_ACTIVE =>, ERR_FLT =>, AUTO_ON =>, TAP_ON =>, TOP_ON =>, MAN_ON =>)
   END_RUNG
   // the same network as SCL:
   "Turntable_DB"();   // "Turntable"
END_REGION

REGION Network 2
   RUNG wire#powerrail
      "stacker_DB"(OFF_SQ :=, INIT_SQ :=, ACK_EF :=, S_PREV :=, S_NEXT :=, SW_AUTO :=, SW_TAP :=, SW_TOP :=, SW_MAN :=, S_SEL :=, S_ON :=, S_OFF :=, T_PUSH :=, S_NO =>, S_MORE =>, S_ACTIVE =>, ERR_FLT =>, AUTO_ON =>, TAP_ON =>, TOP_ON =>, MAN_ON =>)
   END_RUNG
   // the same network as SCL:
   "stacker_DB"();   // "stacker"
END_REGION
END_FUNCTION

FUNCTION "get first free storage" : Void   // FC11, SCL
{ S7_Optimized_Access := 'FALSE' }
VERSION : 0.1
   VAR_OUTPUT
      "target position" : DInt;
   END_VAR
   VAR_TEMP
      i : Int;
      "storage cap" : Int;
   END_VAR
BEGIN
   FOR #i := 1 TO 54 DO
       IF "Storage".status[#i - 1] = FALSE  THEN
           // Statement section IF
           ;
           #"target position" := #i;
           "Storage".status[#i-1] := 1;

           EXIT;
       END_IF;
   END_FOR;

   "Storage"."product type"[#i-1] := "product type";
END_FUNCTION

FUNCTION "Update DB" : Void   // FC12, SCL
{ S7_Optimized_Access := 'FALSE' }
VERSION : 0.1
   VAR_TEMP
      i : Int;
      "storage cap" : Int;
   END_VAR
BEGIN
   "Storage".status["user target position" ] := 0;
   "Storage"."product type"["user target position" ] := 0;
END_FUNCTION

// folder: statistics

FUNCTION "statistics" : Void   // FC13, LAD
{ S7_Optimized_Access := 'FALSE' }
VERSION : 0.1
BEGIN

REGION Network 1
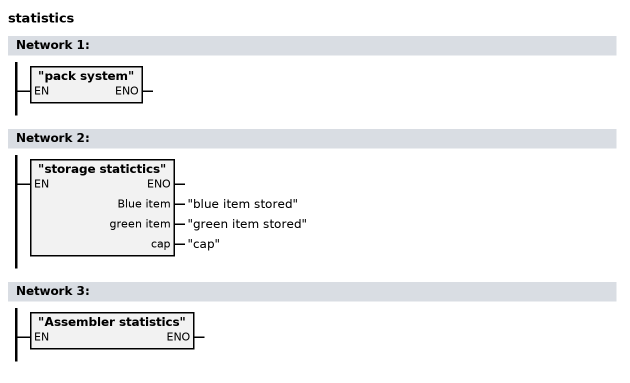
   RUNG wire#powerrail
      "pack system"()
   END_RUNG
   // the same network as SCL:
   "pack system"();
END_REGION

REGION Network 2
   RUNG wire#powerrail
      "storage statictics"("Blue item" => "blue item stored", "green item" => "green item stored", cap => "cap")
   END_RUNG
   // the same network as SCL:
   "storage statictics"("Blue item" => "blue item stored", "green item" => "green item stored", cap => "cap");
END_REGION

REGION Network 3
   RUNG wire#powerrail
      "Assembler statistics"()
   END_RUNG
   // the same network as SCL:
   "Assembler statistics"();
END_REGION
END_FUNCTION

FUNCTION "pack system" : Void   // FC14, LAD
{ S7_Optimized_Access := 'FALSE' }
VERSION : 0.1
   VAR_TEMP   // added for the SCL form of the ladder/FBD networks
      _s5time1 : S5Time;
   END_VAR
BEGIN

REGION Network 1: pick and place UptimeGreen
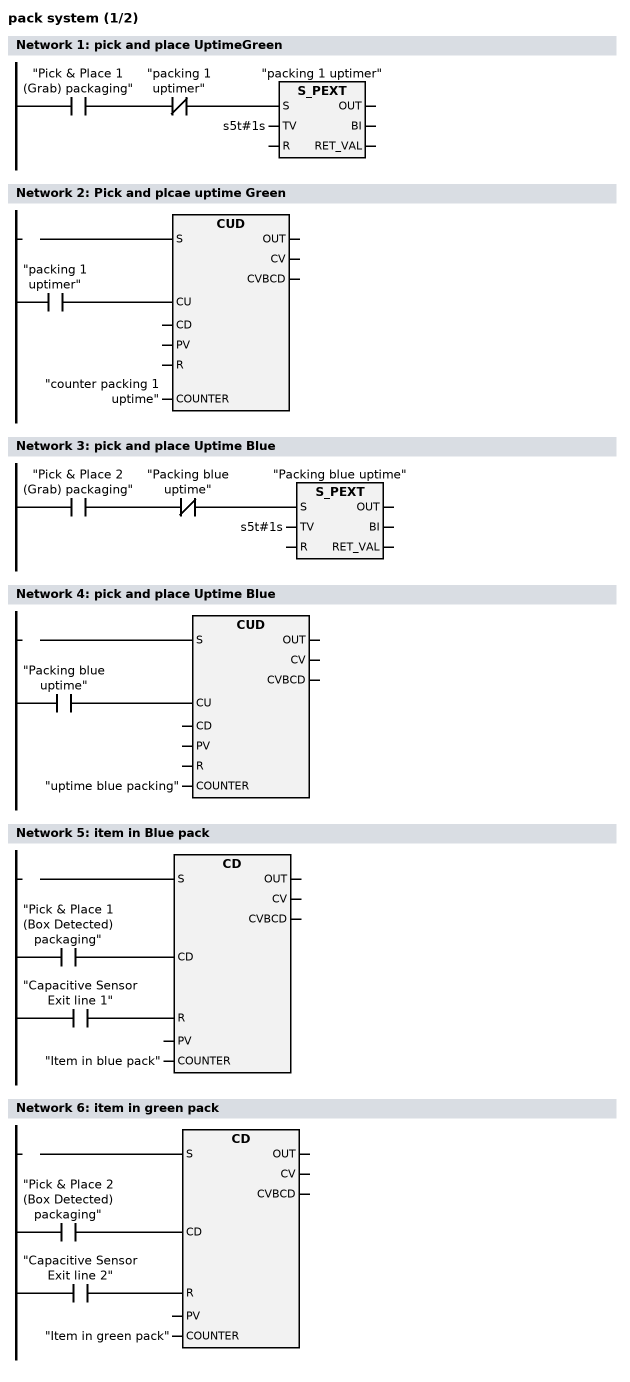
   RUNG wire#powerrail
      Contact( "Pick & Place 1 (Grab) packaging" )
      I_Contact( "packing 1 uptimer" )
      S_PEXT(T_NO := "packing 1 uptimer", TV := s5t#1s, R :=, BI =>, RET_VAL =>)
   END_RUNG
   // the same network as SCL:
   #_s5time1 := S_PEXT(T_NO := "packing 1 uptimer",
                       S := "Pick & Place 1 (Grab) packaging" AND NOT "packing 1 uptimer",
                       TV := s5t#1s);
END_REGION

REGION Network 2: Pick and plcae uptime Green
   // no SCL statement known for Cud: written as a call
   Cud(cu := "packing 1 uptimer", "counter" := "counter packing 1 uptime");
END_REGION

REGION Network 3: pick and place Uptime Blue
   RUNG wire#powerrail
      Contact( "Pick & Place 2 (Grab) packaging" )
      I_Contact( "Packing blue uptime" )
      S_PEXT(T_NO := "Packing blue uptime", TV := s5t#1s, R :=, BI =>, RET_VAL =>)
   END_RUNG
   // the same network as SCL:
   #_s5time1 := S_PEXT(T_NO := "Packing blue uptime",
                       S := "Pick & Place 2 (Grab) packaging" AND NOT "Packing blue uptime",
                       TV := s5t#1s);
END_REGION

REGION Network 4: pick and place Uptime Blue
   // no SCL statement known for Cud: written as a call
   Cud(cu := "Packing blue uptime", "counter" := "uptime blue packing");
END_REGION

REGION Network 5: item in Blue pack
   // no SCL statement known for Cd: written as a call
   Cd(cd := "Pick & Place 1 (Box Detected) packaging",
      r := "Capacitive Sensor Exit line 1",
      "counter" := "Item in blue pack");
END_REGION

REGION Network 6: item in green pack
   // no SCL statement known for Cd: written as a call
   Cd(cd := "Pick & Place 2 (Box Detected) packaging",
      r := "Capacitive Sensor Exit line 2",
      "counter" := "Item in green pack");
END_REGION

REGION Network 7: Blue pack produced
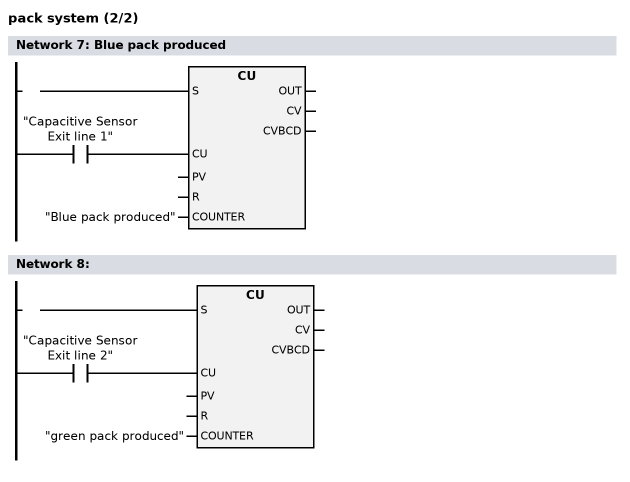
   // no SCL statement known for Cu: written as a call
   Cu(cu := "Capacitive Sensor Exit line 1", "counter" := "Blue pack produced");
END_REGION

REGION Network 8
   // no SCL statement known for Cu: written as a call
   Cu(cu := "Capacitive Sensor Exit line 2", "counter" := "green pack produced");
END_REGION
END_FUNCTION

FUNCTION "storage statictics" : Void   // FC15, SCL
{ S7_Optimized_Access := 'FALSE' }
VERSION : 0.1
   VAR_OUTPUT
      "Blue item" : Int;
      "green item" : Int;
      cap : Int;
   END_VAR
   VAR_TEMP
      i : Int;
   END_VAR
BEGIN
   #"green item" := 0;
   #"Blue item" := 0;
   #cap := 0;
   FOR #i := 0 TO 53 DO
       // Statement section FOR
       // 


       IF "Storage"."product type"[#i] = 2 THEN
           #"Blue item" := #"Blue item" + 1;
           // Statement section IF
           ;
       END_IF;
       IF "Storage"."product type"[#i] =0 THEN
           // Statement section IF
           ;
           #cap := #cap+1;
       END_IF;
       IF "Storage"."product type"[#i] = 1 THEN
           // Statement section IF
           ;
           #"green item" := #"green item" + 1;
       END_IF;



       ;
   END_FOR;
   #cap := #cap + 1;
END_FUNCTION

FUNCTION "Assembler statistics" : Void   // FC16, LAD
{ S7_Optimized_Access := 'FALSE' }
VERSION : 0.1
   VAR_TEMP   // added for the SCL form of the ladder/FBD networks
      _s5time1 : S5Time;
   END_VAR
BEGIN

REGION Network 1: Blue product manufactored
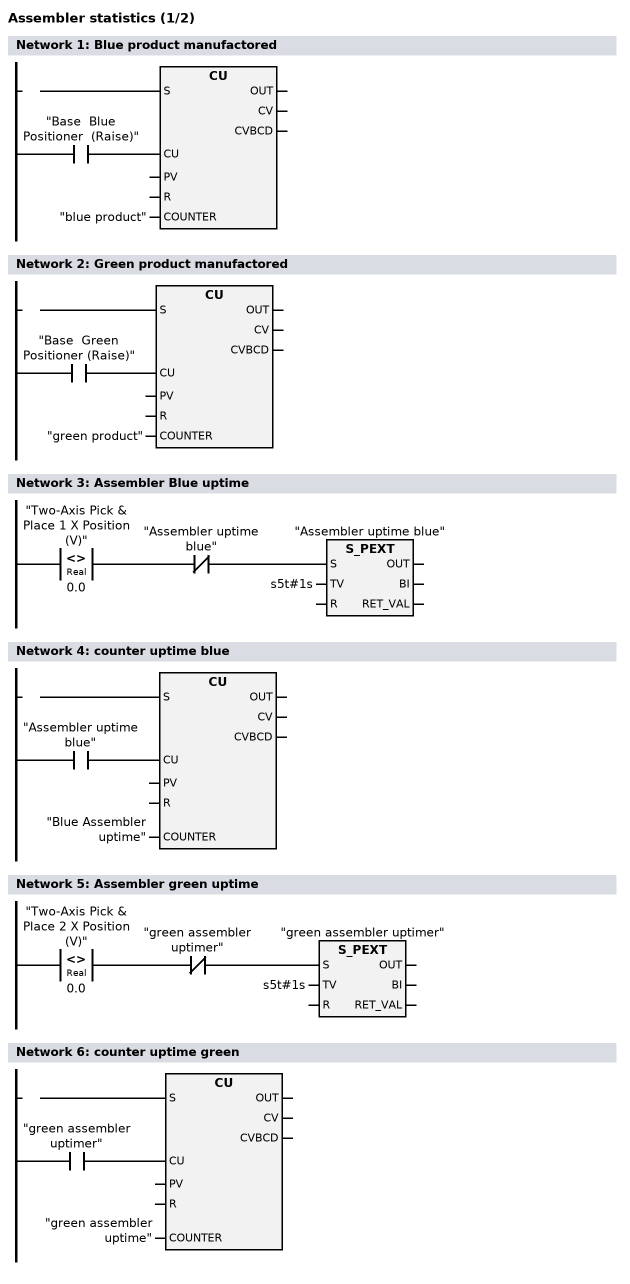
   // no SCL statement known for Cu: written as a call
   Cu(cu := "Base  Blue Positioner  (Raise)", "counter" := "blue product");
END_REGION

REGION Network 2: Green product manufactored
   // no SCL statement known for Cu: written as a call
   Cu(cu := "Base  Green Positioner (Raise)", "counter" := "green product");
END_REGION

REGION Network 3: Assembler Blue uptime
   RUNG wire#powerrail
      { S7_Templates := "SrcType := Real" } NE_Contact(in1 := "Two-Axis Pick & Place 1 X Position (V)", in2 := 0.0)
      I_Contact( "Assembler uptime blue" )
      S_PEXT(T_NO := "Assembler uptime blue", TV := s5t#1s, R :=, BI =>, RET_VAL =>)
   END_RUNG
   // the same network as SCL:
   #_s5time1 := S_PEXT(T_NO := "Assembler uptime blue",
                       S := ("Two-Axis Pick & Place 1 X Position (V)" <> 0.0) AND NOT "Assembler uptime blue",
                       TV := s5t#1s);
END_REGION

REGION Network 4: counter uptime blue
   // no SCL statement known for Cu: written as a call
   Cu(cu := "Assembler uptime blue", "counter" := "Blue Assembler uptime");
END_REGION

REGION Network 5: Assembler green uptime
   RUNG wire#powerrail
      { S7_Templates := "SrcType := Real" } NE_Contact(in1 := "Two-Axis Pick & Place 2 X Position (V)", in2 := 0.0)
      I_Contact( "green assembler uptimer" )
      S_PEXT(T_NO := "green assembler uptimer", TV := s5t#1s, R :=, BI =>, RET_VAL =>)
   END_RUNG
   // the same network as SCL:
   #_s5time1 := S_PEXT(T_NO := "green assembler uptimer",
                       S := ("Two-Axis Pick & Place 2 X Position (V)" <> 0.0) AND NOT "green assembler uptimer",
                       TV := s5t#1s);
END_REGION

REGION Network 6: counter uptime green
   // no SCL statement known for Cu: written as a call
   Cu(cu := "green assembler uptimer", "counter" := "green assembler uptime");
END_REGION

REGION Network 7: main convoyer uptime
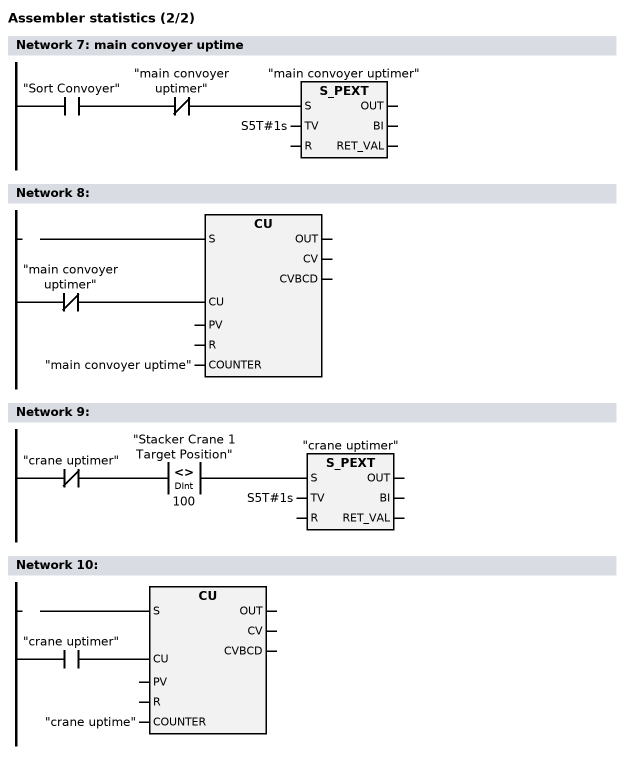
   RUNG wire#powerrail
      Contact( "Sort Convoyer" )
      I_Contact( "main convoyer uptimer" )
      S_PEXT(T_NO := "main convoyer uptimer", TV := S5T#1s, R :=, BI =>, RET_VAL =>)
   END_RUNG
   // the same network as SCL:
   #_s5time1 := S_PEXT(T_NO := "main convoyer uptimer",
                       S := "Sort Convoyer" AND NOT "main convoyer uptimer",
                       TV := S5T#1s);
END_REGION

REGION Network 8
   // no SCL statement known for Cu: written as a call
   Cu(cu := NOT "main convoyer uptimer", "counter" := "main convoyer uptime");
END_REGION

REGION Network 9
   RUNG wire#powerrail
      I_Contact( "crane uptimer" )
      { S7_Templates := "SrcType := DInt" } NE_Contact(in1 := "Stacker Crane 1 Target Position", in2 := 100)
      S_PEXT(T_NO := "crane uptimer", TV := S5T#1s, R :=, BI =>, RET_VAL =>)
   END_RUNG
   // the same network as SCL:
   #_s5time1 := S_PEXT(T_NO := "crane uptimer",
                       S := NOT "crane uptimer" AND ("Stacker Crane 1 Target Position" <> 100),
                       TV := S5T#1s);
END_REGION

REGION Network 10
   // no SCL statement known for Cu: written as a call
   Cu(cu := "crane uptimer", "counter" := "crane uptime");
END_REGION
END_FUNCTION

(* ===== HMI "HMI_RT_1" =====
system functions are stored by id; their names below are inferred from use
connection "HMI_Connection_1": ETHERNET, SIMATIC S7 300/400 MPI

HMI tags "Default tag table"
   "Tag_ScreenNumber" : UInt, internal
   "Sort Convoyer" : Bool = PLC "Sort Convoyer" AT %Q6.7, 1 s
   "Blue Pusher Lid" : Bool = PLC "Blue Pusher Lid" AT %Q1.4, 1 s
   "Blue Pusher Base" : Bool = PLC "Blue Pusher Base" AT %Q1.3, 1 s
   "Assemble Lid Blue Convoyer" : Bool = PLC "Assemble Lid Blue Convoyer" AT %Q0.3, 1 s
   "Assemble Base Blue Convoyer" : Bool = PLC "Assemble Base Blue Convoyer" AT %Q0.1, 1 s
   "Green Pusher Lid" : Bool = PLC "Green Pusher Lid" AT %Q2.0, 1 s
   "Green Pusher Base" : Bool = PLC "Green Pusher Base" AT %Q1.7, 1 s
   "Base  Blue Positioner (Clamp)" : Bool = PLC "Base  Blue Positioner (Clamp)" AT %Q0.6, 1 s
   "Lid  Blue Positioner (Clamp)" : Bool = PLC "Lid  Blue Positioner (Clamp)" AT %Q2.2, 1 s
   "Lid  Green Positioner (Clamp)" : Bool = PLC "Lid  Green Positioner (Clamp)" AT %Q2.3, 1 s
   "Packaging Blue Convoyer" : Bool = PLC "Packaging Blue Convoyer" AT %Q4.1, 1 s
   "Packaging Blue Exit Convoyer 1" : Bool = PLC "Packaging Blue Exit Convoyer 1" AT %Q4.2, 1 s
   "Packaging Blue(Clamp)" : Bool = PLC "Packaging Blue(Clamp)" AT %Q4.5, 1 s
   "Packaging Blue Palet Sensor" : Bool = PLC "Packaging Blue Palet Sensor" AT %I3.3, 1 s
   "initial assembler 1" : Bool = PLC "initial assembler 1" AT %M6.6, 1 s
   "initial assembler 2" : Bool = PLC "initial assembler 2" AT %M6.7, 1 s
   "Storage_status{0}" : Bool = PLC Storage.status[0] AT %DB6.DBX0.0, 1 s
   "Storage_product type{0}" : Int = PLC Storage."product type"[0] AT %DB6.DBW10, 1 s
   "user target position" : DInt = PLC "user target position" AT %MD20, 1 s
   "deploy" : Bool = PLC deploy AT %M10.4, 1 s
   "Storage_product type{2}" : Int = PLC Storage."product type"[2] AT %DB6.DBW14, 1 s
   "Storage_product type{1}" : Int = PLC Storage."product type"[1] AT %DB6.DBW12, 1 s
   "storage" : Array [0..53] of Int = PLC Storage."product type" AT %DB6.DBX10.0, 1 s
   "Storage_cap" : Int = PLC Storage.cap AT %DB6.DBW8, 1 s
   "counter packing 1 uptime" : Counter = PLC "counter packing 1 uptime" AT %C6, 1 s
   "uptime blue packing" : Counter = PLC "uptime blue packing" AT %C7, 1 s
   "Item in blue pack" : Counter = PLC "Item in blue pack" AT %C8, 1 s
   "Item in green pack" : Counter = PLC "Item in green pack" AT %C9, 1 s
   "green pack produced" : Counter = PLC "green pack produced" AT %C11, 1 s
   "Blue pack produced" : Counter = PLC "Blue pack produced" AT %C10, 1 s
   "entry convoyer packing green ready" : Bool = PLC "entry convoyer packing green ready" AT %M9.6, 1 s
   "exit convoyer packing green ready" : Bool = PLC "exit convoyer packing green ready" AT %M10.0, 1 s
   "ready to pack 2" : Bool = PLC "ready to pack 2" AT %M9.0, 1 s
   "reset packer 2" : Bool = PLC "reset packer 2" AT %M9.2, 1 s
   "reset packer 1" : Bool = PLC "reset packer 1" AT %M9.1, 1 s
   "entry convoyer packing blue ready" : Bool = PLC "entry convoyer packing blue ready" AT %M8.4, 1 s
   "exit convoyer packing blue ready" : Bool = PLC "exit convoyer packing blue ready" AT %M8.3, 1 s
   "blue item stored" : Int = PLC "blue item stored" AT %MW26, 1 s
   "green item stored" : Int = PLC "green item stored" AT %MW28, 1 s
   "Load to storage" : Bool = PLC "Load to storage" AT %M10.2, 1 s
   "cap" : Int = PLC cap AT %MW30, 1 s
   "Packaging Green Exit Convoyer" : Bool = PLC "Packaging Green Exit Convoyer" AT %Q5.1, 1 s
   "Packaging Green Convoyer" : Bool = PLC "Packaging Green Convoyer" AT %Q5.0, 1 s
   "Packaging Green (Clamp)" : Bool = PLC "Packaging Green (Clamp)" AT %Q4.6, 1 s
   "blue product" : Counter = PLC "blue product" AT %C12, 1 s
   "green product" : Counter = PLC "green product" AT %C13, 1 s
   "Blue Assembler uptime" : Counter = PLC "Blue Assembler uptime" AT %C14, 1 s
   "green assembler uptime" : Counter = PLC "green assembler uptime" AT %C15, 1 s
   "main convoyer uptime" : Counter = PLC "main convoyer uptime" AT %C16, 1 s
   "start_mach_entry_conv" : Bool = PLC start_mach_entry_conv AT %M0.0, 1 s
   "crane uptime" : Counter = PLC "crane uptime" AT %C17, 1 s

screen "Root screen" 1280x740, template "Template_1"
   on GenerateScreen: SetTag("Tag_ScreenNumber", 1)
   IOField "I/O field_3" at 1210,69 size 40x32; FormatPattern 99
      ProcessValue <- "cap"
   TextField "Text field_1" at 1027,72 size 177x25; Text 'Storage capacity :'
   TextField "Text field_2" at 1027,132 size 177x25; Text 'Blue pack stored :'
   IOField "I/O field_4" at 1210,131 size 40x32; FormatPattern 99
      ProcessValue <- "blue item stored"
   TextField "Text field_3" at 1027,192 size 189x25; Text 'green pack stored :'
   IOField "I/O field_5" at 1210,192 size 40x32; FormatPattern 99
      ProcessValue <- "green item stored"
   Button "HmiScreenItemData" at 36,36 size 159x47; TextOff 'Assembler'; PictureOff "Navigates to Assembler for TP1200 Comfort 17.0.0.0"; PictureOn "Navigates to Assembler for TP1200 Comfort 17.0.0.0"
      on Release: ActivateScreen("Assembler", 0)
   Button "HmiScreenItemData_1" at 36,95 size 159x47; TextOff 'Storage'; PictureOff "Navigates to Storage for TP1200 Comfort 17.0.0.0"; PictureOn "Navigates to Storage for TP1200 Comfort 17.0.0.0"
      on Release: ActivateScreen("Storage", 0)
   Button "HmiScreenItemData_2" at 36,154 size 159x47; TextOff 'Packing'; TextOn 'packing'; PictureOff "Navigates to packing for TP1200 Comfort 17.0.0.0"; PictureOn "Navigates to packing for TP1200 Comfort 17.0.0.0"
      on Release: ActivateScreen("packing", 0)
   Button "HmiScreenItemData_5" at 36,214 size 159x47; TextOff 'System screens'; PictureOff "Navigates to System screens for TP1200 Comfort 17.0.0.0"; PictureOn "Navigates to System screens for TP1200 Comfort 17.0.0.0"
      on Release: ActivateScreen("System screens", 0)
   AlarmView "Alarm view_1" at 213,310 size 1046x348
   TextField "Text field_5" at 291,74 size 277x25; Text 'manufactured blue product :'
   TextField "Text field_6" at 291,130 size 290x25; Text 'manufactured green product :'
   IOField "I/O field_1" at 558,70 size 86x32; FormatPattern 99999
      ProcessValue <- "blue product"
   IOField "I/O field_2" at 558,127 size 86x32; FormatPattern 99999
      ProcessValue <- "green product"
   TextField "Text field_4" at 208,10 size 198x29; Text 'System overview'
   Group "Group" at 1027,69 size 223x155
   TextField "Text field_7" at 665,72 size 217x25; Text 'green pack produced :'
   TextField "Text field_8" at 669,133 size 204x25; Text 'blue pack produced :'
   IOField "I/O field_6" at 875,71 size 96x32; FormatPattern 99999
      ProcessValue <- "green pack produced"
   IOField "I/O field_7" at 875,128 size 96x32; FormatPattern 99999
      ProcessValue <- "Blue pack produced"
   TextField "Text field_9" at 213,274 size 93x29; Text 'Alarms:'
   Switch "Switch_1" at 37,293 size 155x88; CaptionText 'Machining Center'; TextOff 'OFF'; TextOn 'ON'
      ProcessValue <- "start_mach_entry_conv"

Template "Template_1" 1280x740
   Button "Exit" at 1200,679 size 78x59; TextOff 'Exit'; PictureOff "ExitRuntime_TP1200_Comfort_TR"; PictureOn "ExitRuntime_TP1200_Comfort_TR"
      on Release: StopRuntime(0)
   Button "Template_Button" at 1120,679 size 78x59; TextOff 'Text'
   Button "Template_Button_1" at 1040,679 size 78x59; TextOff 'Text'
   Button "Template_Button_2" at 960,679 size 78x59; TextOff 'Text'
   Button "Template_Button_3" at 880,679 size 78x59; TextOff 'Text'
   Button "Template_Button_4" at 800,679 size 78x59; TextOff 'Text'
   Button "Template_Button_5" at 720,679 size 78x59; TextOff 'Text'
   Button "Template_Button_6" at 640,679 size 78x59; TextOff 'Text'
   Button "Template_Button_7" at 561,679 size 78x59; TextOff 'Text'
   Button "Template_Button_8" at 481,679 size 78x59; TextOff 'Text'
   Button "Template_Button_9" at 401,679 size 78x59; TextOff 'Text'
   Button "Template_Button_10" at 321,679 size 78x59; TextOff 'Text'
   Button "Template_Button_11" at 241,679 size 78x59; TextOff 'Text'
   Button "Template_Button_12" at 161,679 size 78x59; TextOff 'Text'
   Button "Template_Button_13" at 81,679 size 78x59; TextOff 'Text'
   Button "Start screen" at 1,679 size 78x59; TextOff 'Start screen'; PictureOff "NavigateHome_TP1200_Comfort_TR"; PictureOn "NavigateHome_TP1200_Comfort_TR"
      on Release: ActivateScreen("Root screen", 0)

screen "Assembler" 1280x740, template "Template_1"
   on GenerateScreen: SetTag("Tag_ScreenNumber", 2)
   Button "Back" at 1,1 size 159x47; TextOff 'Back'
      on Release: ActivateScreen("Root screen", 0)
   Rectangle "Rectangle_1" at 51,311 size 525x48
      Appearance <- "Sort Convoyer"
   Circle "Circle_1" at 105,369 size 33x33
      Appearance <- "Blue Pusher Lid"
   TextField "Text field_1" at 109,391 size 22x131; Text 'Pusher blue lid'
   Rectangle "Rectangle_2" at 85,158 size 69x153
      Appearance <- "Assemble Lid Blue Convoyer"
   Rectangle "Rectangle_3" at 216,128 size 69x183
      Appearance <- "Assemble Base Blue Convoyer"
   Circle "Circle_2" at 234,369 size 33x33
      Appearance <- "Blue Pusher Base"
   TextField "Text field_2" at 238,391 size 22x148; Text 'Pusher blue base'
   Circle "Circle_3" at 386,369 size 33x33
      Appearance <- "Green Pusher Lid"
   TextField "Text field_3" at 390,391 size 22x143; Text 'Pusher green lid'
   Circle "Circle_4" at 515,369 size 33x33
      Appearance <- "Green Pusher Base"
   TextField "Text field_4" at 519,391 size 22x160; Text 'Pusher green base'
   TextField "Text field_5" at 822,137 size 277x25; Text 'manufactured blue product :'
   TextField "Text field_6" at 822,193 size 277x25; Text 'manufactured green product :'
   TextField "Text field_7" at 822,249 size 277x25; Text 'Assembler blue uptime :'
   TextField "Text field_8" at 822,305 size 277x25; Text 'Assembler green uptime :'
   TextField "Text field_9" at 822,361 size 277x25; Text 'main conveyor belt uptime:'
   Circle "Circle_5" at 562,189 size 31x31
      Appearance <- "Base  Blue Positioner (Clamp)"
   TextField "Text field_14" at 581,220 size 47x20; Text 'clamp'
   Circle "Circle_6" at 433,189 size 31x31
      Appearance <- "Lid  Green Positioner (Clamp)"
   TextField "Text field_15" at 441,220 size 47x20; Text 'clamp'
   Circle "Circle_7" at 279,189 size 31x31
      Appearance <- "Base  Blue Positioner (Clamp)"
   TextField "Text field_16" at 285,220 size 47x20; Text 'clamp'
   Circle "Circle_8" at 146,189 size 31x31
      Appearance <- "Lid  Blue Positioner (Clamp)"
   TextField "Text field_17" at 157,220 size 47x20; Text 'clamp'
   IOField "I/O field_1" at 1089,133 size 120x32; FormatPattern 99999
      ProcessValue <- "blue product"
   Button "Button_1" at 425,267 size 96x32; TextOff 'Reset'
      on Release: ResetBit("initial assembler 2")
      on Press: SetBit("initial assembler 2")
   Button "Button_2" at 131,270 size 96x32; TextOff 'Reset'
      on Press: SetBit("initial assembler 1")
      on Release: ResetBit("initial assembler 1")
   IOField "I/O field_2" at 1095,189 size 114x32; FormatPattern 99999
      ProcessValue <- "green product"
   IOField "I/O field_3" at 1056,245 size 152x32; FormatPattern 99999
      ProcessValue <- "Blue Assembler uptime"
   IOField "I/O field_4" at 1057,301 size 152x32; FormatPattern 99999
      ProcessValue <- "green assembler uptime"
   IOField "I/O field_5" at 1074,357 size 134x32; FormatPattern 99999
      ProcessValue <- "main convoyer uptime"

